LIN {X 0,Y 312.808,Z 286.335,A -85,B 0,C 180,E1 -15472.26,E2 -15472.26} C_VEL
LIN {X 0,Y 312.679,Z 286.347,A -85,B 0,C 180,E1 -15474.849,E2 -15474.849} C_VEL
LIN {X 0,Y 312.966,Z 286.313,A -85,B 0,C 180,E1 -15478.72,E2 -15478.72} C_VEL
LIN {X 0,Y 312.908,Z 286.323,A -85,B 0,C 180,E1 -15482.581,E2 -15482.581} C_VEL
LIN {X 0,Y 312.829,Z 286.33,A -85,B 0,C 180,E1 -15486.456,E2 -15486.456} C_VEL
LIN {X 0,Y 312.739,Z 286.341,A -85,B 0,C 180,E1 -15489.057,E2 -15489.057} C_VEL
LIN {X 0,Y 312.615,Z 286.358,A -85,B 0,C 180,E1 -15492.998,E2 -15492.998} C_VEL
LIN {X 0,Y 312.562,Z 286.36,A -85,B 0,C 180,E1 -15495.659,E2 -15495.659} C_VEL
LIN {X 0,Y 312.528,Z 286.365,A -85,B 0,C 180,E1 -15499.719,E2 -15499.719} C_VEL
LIN {X 0,Y 312.509,Z 286.369,A -85,B 0,C 180,E1 -15502.781,E2 -15502.781} C_VEL
LIN {X 0,Y 312.484,Z 286.371,A -85,B 0,C 180,E1 -15506.737,E2 -15506.737} C_VEL
LIN {X 0,Y 312.494,Z 286.371,A -85,B 0,C 180,E1 -15509.661,E2 -15509.661} C_VEL
LIN {X 0,Y 312.52,Z 286.369,A -85,B 0,C 180,E1 -15513.694,E2 -15513.694} C_VEL
LIN {X 0,Y 312.51,Z 286.371,A -85,B 0,C 180,E1 -15517.393,E2 -15517.393} C_VEL
LIN {X 0,Y 312.442,Z 286.374,A -85,B 0,C 180,E1 -15520.722,E2 -15520.722} C_VEL
LIN {X 0,Y 312.452,Z 286.375,A -85,B 0,C 180,E1 -15524.215,E2 -15524.215} C_VEL
LIN {X 0,Y 312.458,Z 286.378,A -85,B 0,C 180,E1 -15527.93,E2 -15527.93} C_VEL
LIN {X 0,Y 312.482,Z 286.376,A -85,B 0,C 180,E1 -15531.929,E2 -15531.929} C_VEL
LIN {X 0,Y 312.536,Z 286.367,A -85,B 0,C 180,E1 -15534.224,E2 -15534.224} C_VEL
LIN {X 0,Y 312.508,Z 286.367,A -85,B 0,C 180,E1 -15537.337,E2 -15537.337} C_VEL
LIN {X 0,Y 312.491,Z 286.369,A -85,B 0,C 180,E1 -15541.304,E2 -15541.304} C_VEL
LIN {X 0,Y 312.68,Z 286.545,A -85,B 0,C 180,E1 -15543.7,E2 -15543.7} C_VEL
LIN {X 0,Y 314.175,Z 295.332,A -85,B 0,C 180,E1 -15546.522,E2 -15546.522} C_VEL
LIN {X 0,Y 313.298,Z 305.478,A -85,B 0,C 180,E1 -15549.656,E2 -15549.656} C_VEL
LIN {X 0,Y 312.436,Z 315.736,A -85,B 0,C 180,E1 -15552.789,E2 -15552.789} C_VEL
LIN {X 0,Y 313.543,Z 332.693,A -85,B 0,C 180,E1 -15553.393,E2 -15553.393} C_VEL
LIN {X 0,Y 314.974,Z 349.181,A -85,B 0,C 180,E1 -15553.982,E2 -15553.982} C_VEL
LIN {X 0,Y 313.99,Z 394.354,A -85,B 0,C 180,E1 -15555.542,E2 -15555.542} C_VEL
LIN {X 0,Y 313.569,Z 406.833,A -85,B 0,C 180,E1 -15556.226,E2 -15556.226} C_VEL
LIN {X 0,Y 313.016,Z 417.039,A -85,B 0,C 180,E1 -15557.027,E2 -15557.027} C_VEL
LIN {X 0,Y 312.578,Z 425.178,A -85,B 0,C 180,E1 -15557.834,E2 -15557.834} C_VEL
LIN {X 0,Y 312.139,Z 433.195,A -85,B 0,C 180,E1 -15558.805,E2 -15558.805} C_VEL
LIN {X 0,Y 311.741,Z 441.983,A -85,B 0,C 180,E1 -15560.104,E2 -15560.104} C_VEL
LIN {X 0,Y 311.412,Z 449.886,A -85,B 0,C 180,E1 -15561.567,E2 -15561.567} C_VEL
LIN {X 0,Y 311.172,Z 456.813,A -85,B 0,C 180,E1 -15563.192,E2 -15563.192} C_VEL
LIN {X 0,Y 311.051,Z 460.872,A -85,B 0,C 180,E1 -15564.339,E2 -15564.339} C_VEL
LIN {X 0,Y 310.982,Z 464.265,A -85,B 0,C 180,E1 -15565.466,E2 -15565.466} C_VEL
LIN {X 0,Y 310.82,Z 468.668,A -85,B 0,C 180,E1 -15567.41,E2 -15567.41} C_VEL
LIN {X 0,Y 310.924,Z 470.88,A -85,B 0,C 180,E1 -15568.707,E2 -15568.707} C_VEL
LIN {X 0,Y 311.031,Z 472.489,A -85,B 0,C 180,E1 -15570.002,E2 -15570.002} C_VEL
LIN {X 0,Y 310.703,Z 473.409,A -85,B 0,C 180,E1 -15571.298,E2 -15571.298} C_VEL
LIN {X 0,Y 310.703,Z 473.802,A -85,B 0,C 180,E1 -15572.595,E2 -15572.595} C_VEL
LIN {X 0,Y 310.758,Z 473.691,A -85,B 0,C 180,E1 -15573.892,E2 -15573.892} C_VEL
LIN {X 0,Y 310.897,Z 472.45,A -85,B 0,C 180,E1 -15575.902,E2 -15575.902} C_VEL
LIN {X 0,Y 311.304,Z 470.124,A -85,B 0,C 180,E1 -15577.787,E2 -15577.787} C_VEL
LIN {X 0,Y 312.084,Z 466.493,A -85,B 0,C 180,E1 -15579.726,E2 -15579.726} C_VEL
LIN {X 0,Y 313.249,Z 461.354,A -85,B 0,C 180,E1 -15581.651,E2 -15581.651} C_VEL
LIN {X 0,Y 314.485,Z 455.869,A -85,B 0,C 180,E1 -15583.244,E2 -15583.244} C_VEL
LIN {X 0,Y 315.901,Z 449.073,A -85,B 0,C 180,E1 -15584.826,E2 -15584.826} C_VEL
LIN {X 0,Y 317.87,Z 439.738,A -85,B 0,C 180,E1 -15586.541,E2 -15586.541} C_VEL
LIN {X 0,Y 319.594,Z 431.167,A -85,B 0,C 180,E1 -15587.767,E2 -15587.767} C_VEL
LIN {X 0,Y 321.226,Z 422.026,A -85,B 0,C 180,E1 -15588.829,E2 -15588.829} C_VEL
LIN {X 0,Y 323.179,Z 410.428,A -85,B 0,C 180,E1 -15589.866,E2 -15589.866} C_VEL
LIN {X 0,Y 324.712,Z 399.087,A -85,B 0,C 180,E1 -15590.594,E2 -15590.594} C_VEL
LIN {X 0,Y 325.906,Z 386.794,A -85,B 0,C 180,E1 -15591.176,E2 -15591.176} C_VEL
LIN {X 0,Y 328.411,Z 352.215,A -85,B 0,C 180,E1 -15592.473,E2 -15592.473} C_VEL
LIN {X 0,Y 326.923,Z 339.744,A -85,B 0,C 180,E1 -15593.305,E2 -15593.305} C_VEL
LIN {X 0,Y 324.202,Z 325.651,A -85,B 0,C 180,E1 -15594.496,E2 -15594.496} C_VEL
LIN {X 0,Y 321.224,Z 313.546,A -85,B 0,C 180,E1 -15595.703,E2 -15595.703} C_VEL
LIN {X 0,Y 319.041,Z 308.853,A -85,B 0,C 180,E1 -15596.4,E2 -15596.4} C_VEL
LIN {X 0,Y 317.388,Z 301.3,A -85,B 0,C 180,E1 -15599.155,E2 -15599.155} C_VEL
LIN {X 0,Y 315.056,Z 293.728,A -85,B 0,C 180,E1 -15602.371,E2 -15602.371} C_VEL
LIN {X 0,Y 312.535,Z 286.365,A -85,B 0,C 180,E1 -15606.212,E2 -15606.212} C_VEL
LIN {X 0,Y 312.457,Z 286.373,A -85,B 0,C 180,E1 -15610.109,E2 -15610.109} C_VEL
LIN {X 0,Y 312.457,Z 286.374,A -85,B 0,C 180,E1 -15614.211,E2 -15614.211} C_VEL
LIN {X 0,Y 312.446,Z 286.373,A -85,B 0,C 180,E1 -15617.929,E2 -15617.929} C_VEL
LIN {X 0,Y 312.495,Z 286.365,A -85,B 0,C 180,E1 -15621.922,E2 -15621.922} C_VEL
LIN {X 0,Y 312.549,Z 286.361,A -85,B 0,C 180,E1 -15624.217,E2 -15624.217} C_VEL
LIN {X 0,Y 312.521,Z 286.366,A -85,B 0,C 180,E1 -15627.33,E2 -15627.33} C_VEL
LIN {X 0,Y 312.542,Z 286.523,A -85,B 0,C 180,E1 -15629.038,E2 -15629.038} C_VEL
LIN {X 0,Y 314.433,Z 291.517,A -85,B 0,C 180,E1 -15631.525,E2 -15631.525} C_VEL
LIN {X 0,Y 315.715,Z 294.654,A -85,B 0,C 180,E1 -15632.848,E2 -15632.848} C_VEL
LIN {X 0,Y 320.679,Z 302.089,A -85,B 0,C 180,E1 -15634.363,E2 -15634.363} C_VEL
LIN {X 0,Y 325.742,Z 310.91,A -85,B 0,C 180,E1 -15635.813,E2 -15635.813} C_VEL
LIN {X 0,Y 330.204,Z 320.269,A -85,B 0,C 180,E1 -15637.053,E2 -15637.053} C_VEL
LIN {X 0,Y 330.37,Z 321.468,A -85,B 0,C 180,E1 -15637.137,E2 -15637.137} C_VEL
LIN {X 0,Y 326.132,Z 374.77,A -85,B 0,C 180,E1 -15639.166,E2 -15639.166} C_VEL
LIN {X 0,Y 324.812,Z 387.33,A -85,B 0,C 180,E1 -15639.905,E2 -15639.905} C_VEL
LIN {X 0,Y 323.647,Z 396.64,A -85,B 0,C 180,E1 -15640.656,E2 -15640.656} C_VEL
LIN {X 0,Y 322.303,Z 405.621,A -85,B 0,C 180,E1 -15641.562,E2 -15641.562} C_VEL
LIN {X 0,Y 320.632,Z 415.281,A -85,B 0,C 180,E1 -15642.782,E2 -15642.782} C_VEL
LIN {X 0,Y 319.098,Z 422.949,A -85,B 0,C 180,E1 -15644.014,E2 -15644.014} C_VEL
LIN {X 0,Y 317.777,Z 429.28,A -85,B 0,C 180,E1 -15645.26,E2 -15645.26} C_VEL
LIN {X 0,Y 316.19,Z 435.818,A -85,B 0,C 180,E1 -15646.825,E2 -15646.825} C_VEL
LIN {X 0,Y 314.829,Z 441.072,A -85,B 0,C 180,E1 -15648.404,E2 -15648.404} C_VEL
LIN {X 0,Y 313.901,Z 444.428,A -85,B 0,C 180,E1 -15649.676,E2 -15649.676} C_VEL
LIN {X 0,Y 313.26,Z 447.125,A -85,B 0,C 180,E1 -15650.959,E2 -15650.959} C_VEL
LIN {X 0,Y 312.448,Z 449.278,A -85,B 0,C 180,E1 -15652.238,E2 -15652.238} C_VEL
LIN {X 0,Y 311.829,Z 450.845,A -85,B 0,C 180,E1 -15653.523,E2 -15653.523} C_VEL
LIN {X 0,Y 311.53,Z 451.786,A -85,B 0,C 180,E1 -15654.816,E2 -15654.816} C_VEL
LIN {X 0,Y 311.246,Z 452.205,A -85,B 0,C 180,E1 -15656.109,E2 -15656.109} C_VEL
LIN {X 0,Y 310.975,Z 452.125,A -85,B 0,C 180,E1 -15657.403,E2 -15657.403} C_VEL
LIN {X 0,Y 310.798,Z 451.534,A -85,B 0,C 180,E1 -15658.698,E2 -15658.698} C_VEL
LIN {X 0,Y 310.737,Z 450.385,A -85,B 0,C 180,E1 -15659.993,E2 -15659.993} C_VEL
LIN {X 0,Y 310.733,Z 447.533,A -85,B 0,C 180,E1 -15661.938,E2 -15661.938} C_VEL
LIN {X 0,Y 310.866,Z 444.951,A -85,B 0,C 180,E1 -15663.233,E2 -15663.233} C_VEL
LIN {X 0,Y 310.987,Z 441.657,A -85,B 0,C 180,E1 -15664.53,E2 -15664.53} C_VEL
LIN {X 0,Y 311.148,Z 435.238,A -85,B 0,C 180,E1 -15666.478,E2 -15666.478} C_VEL
LIN {X 0,Y 311.464,Z 429.92,A -85,B 0,C 180,E1 -15667.774,E2 -15667.774} C_VEL
LIN {X 0,Y 311.765,Z 423.504,A -85,B 0,C 180,E1 -15669.072,E2 -15669.072} C_VEL
LIN {X 0,Y 312.089,Z 415.727,A -85,B 0,C 180,E1 -15670.372,E2 -15670.372} C_VEL
LIN {X 0,Y 312.707,Z 406.255,A -85,B 0,C 180,E1 -15671.663,E2 -15671.663} C_VEL
LIN {X 0,Y 313.162,Z 395.383,A -85,B 0,C 180,E1 -15672.797,E2 -15672.797} C_VEL
LIN {X 0,Y 313.618,Z 385.414,A -85,B 0,C 180,E1 -15673.602,E2 -15673.602} C_VEL
LIN {X 0,Y 313.997,Z 373.275,A -85,B 0,C 180,E1 -15674.328,E2 -15674.328} C_VEL
LIN {X 0,Y 314.475,Z 353.255,A -85,B 0,C 180,E1 -15675.051,E2 -15675.051} C_VEL
LIN {X 0,Y 315.258,Z 313.185,A -85,B 0,C 180,E1 -15676.405,E2 -15676.405} C_VEL
LIN {X 0,Y 312.719,Z 292.458,A -85,B 0,C 180,E1 -15677.169,E2 -15677.169} C_VEL
LIN {X 0,Y 312.756,Z 286.337,A -85,B 0,C 180,E1 -15679.323,E2 -15679.323} C_VEL
LIN {X 0,Y 312.478,Z 286.373,A -85,B 0,C 180,E1 -15683.873,E2 -15683.873} C_VEL
LIN {X 0,Y 312.468,Z 286.373,A -85,B 0,C 180,E1 -15686.724,E2 -15686.724} C_VEL
LIN {X 0,Y 312.451,Z 286.374,A -85,B 0,C 180,E1 -15689.65,E2 -15689.65} C_VEL
LIN {X 0,Y 312.501,Z 286.368,A -85,B 0,C 180,E1 -15693.681,E2 -15693.681} C_VEL
LIN {X 0,Y 312.491,Z 286.369,A -85,B 0,C 180,E1 -15697.379,E2 -15697.379} C_VEL
LIN {X 0,Y 312.415,Z 286.383,A -85,B 0,C 180,E1 -15700.71,E2 -15700.71} C_VEL
LIN {X 0,Y 312.423,Z 286.379,A -85,B 0,C 180,E1 -15704.203,E2 -15704.203} C_VEL
LIN {X 0,Y 312.437,Z 286.375,A -85,B 0,C 180,E1 -15707.915,E2 -15707.915} C_VEL
LIN {X 0,Y 312.464,Z 286.378,A -85,B 0,C 180,E1 -15710.964,E2 -15710.964} C_VEL
LIN {X 0,Y 312.495,Z 286.368,A -85,B 0,C 180,E1 -15714.213,E2 -15714.213} C_VEL
LIN {X 0,Y 312.463,Z 286.375,A -85,B 0,C 180,E1 -15717.327,E2 -15717.327} C_VEL
LIN {X 0,Y 312.526,Z 286.365,A -85,B 0,C 180,E1 -15721.818,E2 -15721.818} C_VEL
LIN {X 0,Y 312.541,Z 286.363,A -85,B 0,C 180,E1 -15724.705,E2 -15724.705} C_VEL
LIN {X 0,Y 312.522,Z 286.369,A -85,B 0,C 180,E1 -15727.522,E2 -15727.522} C_VEL
LIN {X 0,Y 312.591,Z 286.361,A -85,B 0,C 180,E1 -15731.651,E2 -15731.651} C_VEL
LIN {X 0,Y 312.645,Z 286.354,A -85,B 0,C 180,E1 -15735.682,E2 -15735.682} C_VEL
LIN {X 0,Y 312.652,Z 286.354,A -85,B 0,C 180,E1 -15739.638,E2 -15739.638} C_VEL
LIN {X 0,Y 312.81,Z 286.331,A -85,B 0,C 180,E1 -15742.251,E2 -15742.251} C_VEL
LIN {X 0,Y 312.67,Z 286.346,A -85,B 0,C 180,E1 -15744.839,E2 -15744.839} C_VEL
LIN {X 0,Y 312.908,Z 286.318,A -85,B 0,C 180,E1 -15747.423,E2 -15747.423} C_VEL
LIN {X 0,Y 313.067,Z 286.303,A -85,B 0,C 180,E1 -15749.998,E2 -15749.998} C_VEL
LIN {X 0,Y 312.906,Z 286.318,A -85,B 0,C 180,E1 -15752.572,E2 -15752.572} C_VEL
LIN {X 0,Y 312.849,Z 286.327,A -85,B 0,C 180,E1 -15756.447,E2 -15756.447} C_VEL
LIN {X 0,Y 312.732,Z 286.339,A -85,B 0,C 180,E1 -15759.048,E2 -15759.048} C_VEL
LIN {X 0,Y 312.581,Z 286.358,A -85,B 0,C 180,E1 -15762.991,E2 -15762.991} C_VEL
LIN {X 0,Y 312.575,Z 286.358,A -85,B 0,C 180,E1 -15765.65,E2 -15765.65} C_VEL
LIN {X 0,Y 312.554,Z 286.361,A -85,B 0,C 180,E1 -15769.225,E2 -15769.225} C_VEL
LIN {X 0,Y 312.475,Z 286.375,A -85,B 0,C 180,E1 -15772.782,E2 -15772.782} C_VEL
LIN {X 0,Y 312.544,Z 286.362,A -85,B 0,C 180,E1 -15775.935,E2 -15775.935} C_VEL
LIN {X 0,Y 312.493,Z 286.368,A -85,B 0,C 180,E1 -15779.652,E2 -15779.652} C_VEL
LIN {X 0,Y 312.469,Z 286.372,A -85,B 0,C 180,E1 -15783.692,E2 -15783.692} C_VEL
LIN {X 0,Y 312.492,Z 286.371,A -85,B 0,C 180,E1 -15787.386,E2 -15787.386} C_VEL
LIN {X 0,Y 312.481,Z 286.372,A -85,B 0,C 180,E1 -15790.707,E2 -15790.707} C_VEL
LIN {X 0,Y 312.549,Z 286.361,A -85,B 0,C 180,E1 -15794.188,E2 -15794.188} C_VEL
LIN {X 0,Y 312.513,Z 286.367,A -85,B 0,C 180,E1 -15797.909,E2 -15797.909} C_VEL
LIN {X 0,Y 312.502,Z 286.369,A -85,B 0,C 180,E1 -15801.914,E2 -15801.914} C_VEL
LIN {X 0,Y 312.467,Z 286.375,A -85,B 0,C 180,E1 -15805.795,E2 -15805.795} C_VEL
LIN {X 0,Y 312.483,Z 286.37,A -85,B 0,C 180,E1 -15808.859,E2 -15808.859} C_VEL
LIN {X 0,Y 312.535,Z 286.368,A -85,B 0,C 180,E1 -15811.83,E2 -15811.83} C_VEL
LIN {X 0,Y 312.551,Z 286.361,A -85,B 0,C 180,E1 -15814.717,E2 -15814.717} C_VEL
LIN {X 0,Y 312.499,Z 286.367,A -85,B 0,C 180,E1 -15818.015,E2 -15818.015} C_VEL
LIN {X 0,Y 312.538,Z 286.366,A -85,B 0,C 180,E1 -15821.658,E2 -15821.658} C_VEL
LIN {X 0,Y 312.553,Z 286.36,A -85,B 0,C 180,E1 -15823.623,E2 -15823.623} C_VEL
LIN {X 0,Y 311.906,Z 286.444,A -85,B 0,C 180,E1 -15824.699,E2 -15824.699} C_VEL
LIN {X 0,Y 309.047,Z 286.8,A -85,B 0,C 180,E1 -15826.449,E2 -15826.449} C_VEL
LIN {X 0,Y 306.64,Z 287.1,A -85,B 0,C 180,E1 -15827.869,E2 -15827.869} C_VEL
LIN {X 0,Y 305.652,Z 287.221,A -85,B 0,C 180,E1 -15828.969,E2 -15828.969} C_VEL
LIN {X 0,Y 305.596,Z 287.228,A -85,B 0,C 180,E1 -15829.341,E2 -15829.341} C_VEL
LIN {X 0,Y 305.75,Z 287.212,A -85,B 0,C 180,E1 -15832.08,E2 -15832.08} C_VEL
LIN {X 0,Y 305.649,Z 287.223,A -85,B 0,C 180,E1 -15834.73,E2 -15834.73} C_VEL
LIN {X 0,Y 305.933,Z 287.189,A -85,B 0,C 180,E1 -15838.69,E2 -15838.69} C_VEL
LIN {X 0,Y 305.923,Z 287.187,A -85,B 0,C 180,E1 -15841.323,E2 -15841.323} C_VEL
LIN {X 0,Y 305.652,Z 287.221,A -85,B 0,C 180,E1 -15845.284,E2 -15845.284} C_VEL
LIN {X 0,Y 305.734,Z 287.211,A -85,B 0,C 180,E1 -15847.934,E2 -15847.934} C_VEL
LIN {X 0,Y 305.585,Z 287.229,A -85,B 0,C 180,E1 -15851.952,E2 -15851.952} C_VEL
LIN {X 0,Y 305.551,Z 287.238,A -85,B 0,C 180,E1 -15854.985,E2 -15854.985} C_VEL
LIN {X 0,Y 305.502,Z 287.243,A -85,B 0,C 180,E1 -15858.794,E2 -15858.794} C_VEL
LIN {X 0,Y 305.452,Z 287.25,A -85,B 0,C 180,E1 -15863.032,E2 -15863.032} C_VEL
LIN {X 0,Y 305.45,Z 287.246,A -85,B 0,C 180,E1 -15866.197,E2 -15866.197} C_VEL
LIN {X 0,Y 305.447,Z 287.25,A -85,B 0,C 180,E1 -15869.039,E2 -15869.039} C_VEL
LIN {X 0,Y 305.436,Z 287.248,A -85,B 0,C 180,E1 -15871.959,E2 -15871.959} C_VEL
LIN {X 0,Y 305.461,Z 287.247,A -85,B 0,C 180,E1 -15875.119,E2 -15875.119} C_VEL
LIN {X 0,Y 305.436,Z 287.247,A -85,B 0,C 180,E1 -15878.53,E2 -15878.53} C_VEL
LIN {X 0,Y 305.436,Z 287.247,A -85,B 0,C 180,E1 -15882.586,E2 -15882.586} C_VEL
LIN {X 0,Y 305.424,Z 287.25,A -85,B 0,C 180,E1 -15886.349,E2 -15886.349} C_VEL
LIN {X 0,Y 305.415,Z 287.255,A -85,B 0,C 180,E1 -15889.889,E2 -15889.889} C_VEL
LIN {X 0,Y 305.467,Z 287.246,A -85,B 0,C 180,E1 -15893.642,E2 -15893.642} C_VEL
LIN {X 0,Y 305.472,Z 287.245,A -85,B 0,C 180,E1 -15896.487,E2 -15896.487} C_VEL
LIN {X 0,Y 305.424,Z 287.25,A -85,B 0,C 180,E1 -15899.59,E2 -15899.59} C_VEL
LIN {X 0,Y 305.616,Z 287.307,A -85,B 0,C 180,E1 -15903.638,E2 -15903.638} C_VEL
LIN {X 0,Y 307.022,Z 295.41,A -85,B 0,C 180,E1 -15906.305,E2 -15906.305} C_VEL
LIN {X 0,Y 306.69,Z 301.192,A -85,B 0,C 180,E1 -15908.14,E2 -15908.14} C_VEL
LIN {X 0,Y 305.38,Z 315.452,A -85,B 0,C 180,E1 -15912.636,E2 -15912.636} C_VEL
LIN {X 0,Y 306.378,Z 331.761,A -85,B 0,C 180,E1 -15913.238,E2 -15913.238} C_VEL
LIN {X 0,Y 307.903,Z 349.63,A -85,B 0,C 180,E1 -15913.902,E2 -15913.902} C_VEL
LIN {X 0,Y 306.913,Z 394.247,A -85,B 0,C 180,E1 -15915.498,E2 -15915.498} C_VEL
LIN {X 0,Y 306.468,Z 407.18,A -85,B 0,C 180,E1 -15916.239,E2 -15916.239} C_VEL
LIN {X 0,Y 305.919,Z 417.254,A -85,B 0,C 180,E1 -15917.059,E2 -15917.059} C_VEL
LIN {X 0,Y 305.357,Z 426.75,A -85,B 0,C 180,E1 -15918.048,E2 -15918.048} C_VEL
LIN {X 0,Y 304.903,Z 436.813,A -85,B 0,C 180,E1 -15919.376,E2 -15919.376} C_VEL
LIN {X 0,Y 304.526,Z 444.734,A -85,B 0,C 180,E1 -15920.706,E2 -15920.706} C_VEL
LIN {X 0,Y 304.281,Z 451.287,A -85,B 0,C 180,E1 -15922.037,E2 -15922.037} C_VEL
LIN {X 0,Y 304.097,Z 456.716,A -85,B 0,C 180,E1 -15923.367,E2 -15923.367} C_VEL
LIN {X 0,Y 303.996,Z 461.21,A -85,B 0,C 180,E1 -15924.696,E2 -15924.696} C_VEL
LIN {X 0,Y 303.844,Z 464.871,A -85,B 0,C 180,E1 -15926.023,E2 -15926.023} C_VEL
LIN {X 0,Y 303.808,Z 469.028,A -85,B 0,C 180,E1 -15928.014,E2 -15928.014} C_VEL
LIN {X 0,Y 303.842,Z 470.176,A -85,B 0,C 180,E1 -15928.677,E2 -15928.677} C_VEL
LIN {X 0,Y 303.97,Z 471.84,A -85,B 0,C 180,E1 -15930.002,E2 -15930.002} C_VEL
LIN {X 0,Y 303.622,Z 472.879,A -85,B 0,C 180,E1 -15931.329,E2 -15931.329} C_VEL
LIN {X 0,Y 303.628,Z 473.429,A -85,B 0,C 180,E1 -15932.656,E2 -15932.656} C_VEL
LIN {X 0,Y 303.675,Z 473.472,A -85,B 0,C 180,E1 -15933.983,E2 -15933.983} C_VEL
LIN {X 0,Y 303.792,Z 472.565,A -85,B 0,C 180,E1 -15935.827,E2 -15935.827} C_VEL
LIN {X 0,Y 304.276,Z 470.237,A -85,B 0,C 180,E1 -15937.968,E2 -15937.968} C_VEL
LIN {X 0,Y 305.086,Z 466.811,A -85,B 0,C 180,E1 -15939.951,E2 -15939.951} C_VEL
LIN {X 0,Y 306.341,Z 461.995,A -85,B 0,C 180,E1 -15941.918,E2 -15941.918} C_VEL
LIN {X 0,Y 307.933,Z 455.501,A -85,B 0,C 180,E1 -15943.868,E2 -15943.868} C_VEL
LIN {X 0,Y 309.143,Z 450.242,A -85,B 0,C 180,E1 -15945.158,E2 -15945.158} C_VEL
LIN {X 0,Y 310.569,Z 443.978,A -85,B 0,C 180,E1 -15946.433,E2 -15946.433} C_VEL
LIN {X 0,Y 312.312,Z 436.428,A -85,B 0,C 180,E1 -15947.688,E2 -15947.688} C_VEL
LIN {X 0,Y 314.229,Z 427.283,A -85,B 0,C 180,E1 -15948.925,E2 -15948.925} C_VEL
LIN {X 0,Y 316.098,Z 417.336,A -85,B 0,C 180,E1 -15949.991,E2 -15949.991} C_VEL
LIN {X 0,Y 317.921,Z 406.353,A -85,B 0,C 180,E1 -15950.885,E2 -15950.885} C_VEL
LIN {X 0,Y 319.594,Z 394.24,A -85,B 0,C 180,E1 -15951.615,E2 -15951.615} C_VEL
LIN {X 0,Y 321.622,Z 369.527,A -85,B 0,C 180,E1 -15952.6,E2 -15952.6} C_VEL
LIN {X 0,Y 322.874,Z 353.385,A -85,B 0,C 180,E1 -15953.232,E2 -15953.232} C_VEL
LIN {X 0,Y 321.463,Z 340.839,A -85,B 0,C 180,E1 -15954.132,E2 -15954.132} C_VEL
LIN {X 0,Y 318.87,Z 327.161,A -85,B 0,C 180,E1 -15955.35,E2 -15955.35} C_VEL
LIN {X 0,Y 316.464,Z 317.354,A -85,B 0,C 180,E1 -15956.404,E2 -15956.404} C_VEL
LIN {X 0,Y 314.296,Z 312.894,A -85,B 0,C 180,E1 -15957.128,E2 -15957.128} C_VEL
LIN {X 0,Y 311.945,Z 308.011,A -85,B 0,C 180,E1 -15958.032,E2 -15958.032} C_VEL
LIN {X 0,Y 310.884,Z 303.44,A -85,B 0,C 180,E1 -15959.826,E2 -15959.826} C_VEL
LIN {X 0,Y 308.965,Z 297.154,A -85,B 0,C 180,E1 -15962.68,E2 -15962.68} C_VEL
LIN {X 0,Y 307.021,Z 291.567,A -85,B 0,C 180,E1 -15965.715,E2 -15965.715} C_VEL
LIN {X 0,Y 305.449,Z 287.248,A -85,B 0,C 180,E1 -15968.677,E2 -15968.677} C_VEL
LIN {X 0,Y 305.419,Z 287.253,A -85,B 0,C 180,E1 -15972.572,E2 -15972.572} C_VEL
LIN {X 0,Y 305.421,Z 287.25,A -85,B 0,C 180,E1 -15976.338,E2 -15976.338} C_VEL
LIN {X 0,Y 305.428,Z 287.246,A -85,B 0,C 180,E1 -15979.882,E2 -15979.882} C_VEL
LIN {X 0,Y 305.481,Z 287.24,A -85,B 0,C 180,E1 -15983.634,E2 -15983.634} C_VEL
LIN {X 0,Y 305.486,Z 287.248,A -85,B 0,C 180,E1 -15986.48,E2 -15986.48} C_VEL
LIN {X 0,Y 307.066,Z 291.123,A -85,B 0,C 180,E1 -15988.999,E2 -15988.999} C_VEL
LIN {X 0,Y 308.688,Z 295.341,A -85,B 0,C 180,E1 -15991.171,E2 -15991.171} C_VEL
LIN {X 0,Y 315.081,Z 304.674,A -85,B 0,C 180,E1 -15993.37,E2 -15993.37} C_VEL
LIN {X 0,Y 319.786,Z 312.784,A -85,B 0,C 180,E1 -15994.832,E2 -15994.832} C_VEL
LIN {X 0,Y 324.2,Z 321.551,A -85,B 0,C 180,E1 -15996.13,E2 -15996.13} C_VEL
LIN {X 0,Y 325.013,Z 323.476,A -85,B 0,C 180,E1 -15996.372,E2 -15996.372} C_VEL
LIN {X 0,Y 320.464,Z 375.997,A -85,B 0,C 180,E1 -15998.443,E2 -15998.443} C_VEL
LIN {X 0,Y 319.046,Z 388.238,A -85,B 0,C 180,E1 -15999.188,E2 -15999.188} C_VEL
LIN {X 0,Y 317.797,Z 397.34,A -85,B 0,C 180,E1 -15999.948,E2 -15999.948} C_VEL
LIN {X 0,Y 316.137,Z 407.489,A -85,B 0,C 180,E1 -16001.021,E2 -16001.021} C_VEL
LIN {X 0,Y 314.085,Z 417.682,A -85,B 0,C 180,E1 -16002.412,E2 -16002.412} C_VEL
LIN {X 0,Y 312.509,Z 425.008,A -85,B 0,C 180,E1 -16003.668,E2 -16003.668} C_VEL
LIN {X 0,Y 311.114,Z 431.083,A -85,B 0,C 180,E1 -16004.937,E2 -16004.937} C_VEL
LIN {X 0,Y 309.755,Z 436.186,A -85,B 0,C 180,E1 -16006.212,E2 -16006.212} C_VEL
LIN {X 0,Y 308.565,Z 440.441,A -85,B 0,C 180,E1 -16007.498,E2 -16007.498} C_VEL
LIN {X 0,Y 307,Z 445.503,A -85,B 0,C 180,E1 -16009.441,E2 -16009.441} C_VEL
LIN {X 0,Y 306.322,Z 448.021,A -85,B 0,C 180,E1 -16010.752,E2 -16010.752} C_VEL
LIN {X 0,Y 305.468,Z 450.005,A -85,B 0,C 180,E1 -16012.059,E2 -16012.059} C_VEL
LIN {X 0,Y 304.819,Z 451.444,A -85,B 0,C 180,E1 -16013.374,E2 -16013.374} C_VEL
LIN {X 0,Y 304.479,Z 452.315,A -85,B 0,C 180,E1 -16014.696,E2 -16014.696} C_VEL
LIN {X 0,Y 304.178,Z 452.582,A -85,B 0,C 180,E1 -16016.019,E2 -16016.019} C_VEL
LIN {X 0,Y 303.897,Z 452.339,A -85,B 0,C 180,E1 -16017.342,E2 -16017.342} C_VEL
LIN {X 0,Y 303.712,Z 451.593,A -85,B 0,C 180,E1 -16018.667,E2 -16018.667} C_VEL
LIN {X 0,Y 303.649,Z 450.326,A -85,B 0,C 180,E1 -16019.993,E2 -16019.993} C_VEL
LIN {X 0,Y 303.653,Z 447.255,A -85,B 0,C 180,E1 -16021.983,E2 -16021.983} C_VEL
LIN {X 0,Y 303.898,Z 442.856,A -85,B 0,C 180,E1 -16023.971,E2 -16023.971} C_VEL
LIN {X 0,Y 303.965,Z 436.98,A -85,B 0,C 180,E1 -16025.941,E2 -16025.941} C_VEL
LIN {X 0,Y 304.347,Z 430.388,A -85,B 0,C 180,E1 -16027.623,E2 -16027.623} C_VEL
LIN {X 0,Y 304.632,Z 424.032,A -85,B 0,C 180,E1 -16028.952,E2 -16028.952} C_VEL
LIN {X 0,Y 305.026,Z 416.328,A -85,B 0,C 180,E1 -16030.279,E2 -16030.279} C_VEL
LIN {X 0,Y 305.564,Z 406.898,A -85,B 0,C 180,E1 -16031.603,E2 -16031.603} C_VEL
LIN {X 0,Y 306.042,Z 396.182,A -85,B 0,C 180,E1 -16032.762,E2 -16032.762} C_VEL
LIN {X 0,Y 306.503,Z 386.353,A -85,B 0,C 180,E1 -16033.586,E2 -16033.586} C_VEL
LIN {X 0,Y 306.882,Z 375.278,A -85,B 0,C 180,E1 -16034.287,E2 -16034.287} C_VEL
LIN {X 0,Y 307.226,Z 359.888,A -85,B 0,C 180,E1 -16034.905,E2 -16034.905} C_VEL
LIN {X 0,Y 308.152,Z 313.414,A -85,B 0,C 180,E1 -16036.525,E2 -16036.525} C_VEL
LIN {X 0,Y 305.682,Z 292.925,A -85,B 0,C 180,E1 -16037.304,E2 -16037.304} C_VEL
LIN {X 0,Y 305.714,Z 287.215,A -85,B 0,C 180,E1 -16039.284,E2 -16039.284} C_VEL
LIN {X 0,Y 305.443,Z 287.25,A -85,B 0,C 180,E1 -16044.458,E2 -16044.458} C_VEL
LIN {X 0,Y 305.426,Z 287.249,A -85,B 0,C 180,E1 -16047.391,E2 -16047.391} C_VEL
LIN {X 0,Y 305.4,Z 287.257,A -85,B 0,C 180,E1 -16050.406,E2 -16050.406} C_VEL
LIN {X 0,Y 305.445,Z 287.249,A -85,B 0,C 180,E1 -16054.07,E2 -16054.07} C_VEL
LIN {X 0,Y 305.431,Z 287.252,A -85,B 0,C 180,E1 -16056.735,E2 -16056.735} C_VEL
LIN {X 0,Y 305.384,Z 287.259,A -85,B 0,C 180,E1 -16060.582,E2 -16060.582} C_VEL
LIN {X 0,Y 305.394,Z 287.253,A -85,B 0,C 180,E1 -16063.649,E2 -16063.649} C_VEL
LIN {X 0,Y 305.411,Z 287.251,A -85,B 0,C 180,E1 -16067.41,E2 -16067.41} C_VEL
LIN {X 0,Y 305.426,Z 287.248,A -85,B 0,C 180,E1 -16069.885,E2 -16069.885} C_VEL
LIN {X 0,Y 305.444,Z 287.247,A -85,B 0,C 180,E1 -16073.625,E2 -16073.625} C_VEL
LIN {X 0,Y 305.427,Z 287.25,A -85,B 0,C 180,E1 -16076.476,E2 -16076.476} C_VEL
LIN {X 0,Y 305.439,Z 287.25,A -85,B 0,C 180,E1 -16080.95,E2 -16080.95} C_VEL
LIN {X 0,Y 305.521,Z 287.237,A -85,B 0,C 180,E1 -16084.081,E2 -16084.081} C_VEL
LIN {X 0,Y 305.436,Z 287.247,A -85,B 0,C 180,E1 -16088.396,E2 -16088.396} C_VEL
LIN {X 0,Y 305.533,Z 287.239,A -85,B 0,C 180,E1 -16091.212,E2 -16091.212} C_VEL
LIN {X 0,Y 305.59,Z 287.232,A -85,B 0,C 180,E1 -16095.344,E2 -16095.344} C_VEL
LIN {X 0,Y 305.589,Z 287.231,A -85,B 0,C 180,E1 -16099.396,E2 -16099.396} C_VEL
LIN {X 0,Y 305.753,Z 287.211,A -85,B 0,C 180,E1 -16102.071,E2 -16102.071} C_VEL
LIN {X 0,Y 305.64,Z 287.222,A -85,B 0,C 180,E1 -16104.72,E2 -16104.72} C_VEL
LIN {X 0,Y 305.91,Z 287.189,A -85,B 0,C 180,E1 -16108.681,E2 -16108.681} C_VEL
LIN {X 0,Y 305.91,Z 287.189,A -85,B 0,C 180,E1 -16111.314,E2 -16111.314} C_VEL
LIN {X 0,Y 305.637,Z 287.222,A -85,B 0,C 180,E1 -16115.275,E2 -16115.275} C_VEL
LIN {X 0,Y 305.749,Z 287.212,A -85,B 0,C 180,E1 -16117.925,E2 -16117.925} C_VEL
LIN {X 0,Y 305.551,Z 287.235,A -85,B 0,C 180,E1 -16121.945,E2 -16121.945} C_VEL
LIN {X 0,Y 305.567,Z 287.232,A -85,B 0,C 180,E1 -16125.023,E2 -16125.023} C_VEL
LIN {X 0,Y 305.525,Z 287.24,A -85,B 0,C 180,E1 -16128.784,E2 -16128.784} C_VEL
LIN {X 0,Y 305.434,Z 287.25,A -85,B 0,C 180,E1 -16133.041,E2 -16133.041} C_VEL
LIN {X 0,Y 305.474,Z 287.244,A -85,B 0,C 180,E1 -16136.22,E2 -16136.22} C_VEL
LIN {X 0,Y 305.444,Z 287.25,A -85,B 0,C 180,E1 -16139.052,E2 -16139.052} C_VEL
LIN {X 0,Y 305.415,Z 287.251,A -85,B 0,C 180,E1 -16143.52,E2 -16143.52} C_VEL
LIN {X 0,Y 305.448,Z 287.249,A -85,B 0,C 180,E1 -16146.74,E2 -16146.74} C_VEL
LIN {X 0,Y 305.44,Z 287.248,A -85,B 0,C 180,E1 -16150.61,E2 -16150.61} C_VEL
LIN {X 0,Y 305.499,Z 287.24,A -85,B 0,C 180,E1 -16154.521,E2 -16154.521} C_VEL
LIN {X 0,Y 305.457,Z 287.245,A -85,B 0,C 180,E1 -16158.158,E2 -16158.158} C_VEL
LIN {X 0,Y 305.468,Z 287.248,A -85,B 0,C 180,E1 -16161.607,E2 -16161.607} C_VEL
LIN {X 0,Y 305.423,Z 287.25,A -85,B 0,C 180,E1 -16164.892,E2 -16164.892} C_VEL
LIN {X 0,Y 305.412,Z 287.25,A -85,B 0,C 180,E1 -16168.362,E2 -16168.362} C_VEL
LIN {X 0,Y 305.477,Z 287.243,A -85,B 0,C 180,E1 -16171.119,E2 -16171.119} C_VEL
LIN {X 0,Y 305.537,Z 287.238,A -85,B 0,C 180,E1 -16174.094,E2 -16174.094} C_VEL
LIN {X 0,Y 305.443,Z 287.248,A -85,B 0,C 180,E1 -16178.407,E2 -16178.407} C_VEL
LIN {X 0,Y 305.489,Z 287.241,A -85,B 0,C 180,E1 -16181.219,E2 -16181.219} C_VEL
LIN {X 0,Y 305.601,Z 287.227,A -85,B 0,C 180,E1 -16185.354,E2 -16185.354} C_VEL
LIN {X 0,Y 305.596,Z 287.228,A -85,B 0,C 180,E1 -16189.341,E2 -16189.341} C_VEL
LIN {X 0,Y 305.001,Z 287.306,A -85,B 0,C 180,E1 -16190.443,E2 -16190.443} C_VEL
LIN {X 0,Y 302.193,Z 287.657,A -85,B 0,C 180,E1 -16192.237,E2 -16192.237} C_VEL
LIN {X 0,Y 299.75,Z 287.959,A -85,B 0,C 180,E1 -16193.693,E2 -16193.693} C_VEL
LIN {X 0,Y 298.67,Z 288.092,A -85,B 0,C 180,E1 -16194.82,E2 -16194.82} C_VEL
LIN {X 0,Y 298.568,Z 288.102,A -85,B 0,C 180,E1 -16195.202,E2 -16195.202} C_VEL
LIN {X 0,Y 298.899,Z 288.066,A -85,B 0,C 180,E1 -16198.66,E2 -16198.66} C_VEL
LIN {X 0,Y 298.891,Z 288.063,A -85,B 0,C 180,E1 -16201.354,E2 -16201.354} C_VEL
LIN {X 0,Y 298.621,Z 288.096,A -85,B 0,C 180,E1 -16205.408,E2 -16205.408} C_VEL
LIN {X 0,Y 298.697,Z 288.092,A -85,B 0,C 180,E1 -16208.826,E2 -16208.826} C_VEL
LIN {X 0,Y 298.534,Z 288.108,A -85,B 0,C 180,E1 -16212.238,E2 -16212.238} C_VEL
LIN {X 0,Y 298.516,Z 288.113,A -85,B 0,C 180,E1 -16215.157,E2 -16215.157} C_VEL
LIN {X 0,Y 298.432,Z 288.121,A -85,B 0,C 180,E1 -16219.621,E2 -16219.621} C_VEL
LIN {X 0,Y 298.378,Z 288.128,A -85,B 0,C 180,E1 -16223.61,E2 -16223.61} C_VEL
LIN {X 0,Y 298.401,Z 288.125,A -85,B 0,C 180,E1 -16226.589,E2 -16226.589} C_VEL
LIN {X 0,Y 298.392,Z 288.127,A -85,B 0,C 180,E1 -16229.65,E2 -16229.65} C_VEL
LIN {X 0,Y 298.393,Z 288.125,A -85,B 0,C 180,E1 -16232.806,E2 -16232.806} C_VEL
LIN {X 0,Y 298.404,Z 288.125,A -85,B 0,C 180,E1 -16236.078,E2 -16236.078} C_VEL
LIN {X 0,Y 298.376,Z 288.132,A -85,B 0,C 180,E1 -16239.497,E2 -16239.497} C_VEL
LIN {X 0,Y 298.372,Z 288.128,A -85,B 0,C 180,E1 -16243.102,E2 -16243.102} C_VEL
LIN {X 0,Y 298.374,Z 288.127,A -85,B 0,C 180,E1 -16246.919,E2 -16246.919} C_VEL
LIN {X 0,Y 298.391,Z 288.125,A -85,B 0,C 180,E1 -16251.016,E2 -16251.016} C_VEL
LIN {X 0,Y 298.41,Z 288.128,A -85,B 0,C 180,E1 -16253.932,E2 -16253.932} C_VEL
LIN {X 0,Y 298.4,Z 288.124,A -85,B 0,C 180,E1 -16257.204,E2 -16257.204} C_VEL
LIN {X 0,Y 298.439,Z 288.122,A -85,B 0,C 180,E1 -16261.905,E2 -16261.905} C_VEL
LIN {X 0,Y 298.594,Z 288.276,A -85,B 0,C 180,E1 -16263.657,E2 -16263.657} C_VEL
LIN {X 0,Y 300.005,Z 296.834,A -85,B 0,C 180,E1 -16266.534,E2 -16266.534} C_VEL
LIN {X 0,Y 299.033,Z 307.031,A -85,B 0,C 180,E1 -16269.839,E2 -16269.839} C_VEL
LIN {X 0,Y 298.309,Z 315.184,A -85,B 0,C 180,E1 -16272.478,E2 -16272.478} C_VEL
LIN {X 0,Y 299.273,Z 331.823,A -85,B 0,C 180,E1 -16273.126,E2 -16273.126} C_VEL
LIN {X 0,Y 300.815,Z 349.751,A -85,B 0,C 180,E1 -16273.809,E2 -16273.809} C_VEL
LIN {X 0,Y 299.812,Z 394.099,A -85,B 0,C 180,E1 -16275.45,E2 -16275.45} C_VEL
LIN {X 0,Y 299.404,Z 406.413,A -85,B 0,C 180,E1 -16276.167,E2 -16276.167} C_VEL
LIN {X 0,Y 298.897,Z 415.678,A -85,B 0,C 180,E1 -16276.922,E2 -16276.922} C_VEL
LIN {X 0,Y 298.466,Z 423.95,A -85,B 0,C 180,E1 -16277.767,E2 -16277.767} C_VEL
LIN {X 0,Y 298.025,Z 432.038,A -85,B 0,C 180,E1 -16278.784,E2 -16278.784} C_VEL
LIN {X 0,Y 297.692,Z 439.858,A -85,B 0,C 180,E1 -16279.976,E2 -16279.976} C_VEL
LIN {X 0,Y 297.295,Z 448.087,A -85,B 0,C 180,E1 -16281.506,E2 -16281.506} C_VEL
LIN {X 0,Y 297.058,Z 455.277,A -85,B 0,C 180,E1 -16283.209,E2 -16283.209} C_VEL
LIN {X 0,Y 296.953,Z 459.964,A -85,B 0,C 180,E1 -16284.57,E2 -16284.57} C_VEL
LIN {X 0,Y 296.798,Z 463.821,A -85,B 0,C 180,E1 -16285.929,E2 -16285.929} C_VEL
LIN {X 0,Y 296.69,Z 466.932,A -85,B 0,C 180,E1 -16287.287,E2 -16287.287} C_VEL
LIN {X 0,Y 296.802,Z 469.354,A -85,B 0,C 180,E1 -16288.645,E2 -16288.645} C_VEL
LIN {X 0,Y 296.909,Z 471.149,A -85,B 0,C 180,E1 -16290.002,E2 -16290.002} C_VEL
LIN {X 0,Y 296.542,Z 472.348,A -85,B 0,C 180,E1 -16291.36,E2 -16291.36} C_VEL
LIN {X 0,Y 296.556,Z 473.054,A -85,B 0,C 180,E1 -16292.719,E2 -16292.719} C_VEL
LIN {X 0,Y 296.594,Z 473.23,A -85,B 0,C 180,E1 -16294.079,E2 -16294.079} C_VEL
LIN {X 0,Y 296.685,Z 472.66,A -85,B 0,C 180,E1 -16295.746,E2 -16295.746} C_VEL
LIN {X 0,Y 297.233,Z 470.364,A -85,B 0,C 180,E1 -16298.158,E2 -16298.158} C_VEL
LIN {X 0,Y 298.106,Z 467.102,A -85,B 0,C 180,E1 -16300.187,E2 -16300.187} C_VEL
LIN {X 0,Y 298.944,Z 464.22,A -85,B 0,C 180,E1 -16301.529,E2 -16301.529} C_VEL
LIN {X 0,Y 300.544,Z 458.677,A -85,B 0,C 180,E1 -16303.526,E2 -16303.526} C_VEL
LIN {X 0,Y 302.392,Z 451.465,A -85,B 0,C 180,E1 -16305.504,E2 -16305.504} C_VEL
LIN {X 0,Y 304.318,Z 443.736,A -85,B 0,C 180,E1 -16307.127,E2 -16307.127} C_VEL
LIN {X 0,Y 306.16,Z 436.315,A -85,B 0,C 180,E1 -16308.401,E2 -16308.401} C_VEL
LIN {X 0,Y 308.511,Z 426.101,A -85,B 0,C 180,E1 -16309.809,E2 -16309.809} C_VEL
LIN {X 0,Y 310.54,Z 415.838,A -85,B 0,C 180,E1 -16310.884,E2 -16310.884} C_VEL
LIN {X 0,Y 312.31,Z 405.63,A -85,B 0,C 180,E1 -16311.711,E2 -16311.711} C_VEL
LIN {X 0,Y 314.214,Z 392.445,A -85,B 0,C 180,E1 -16312.49,E2 -16312.49} C_VEL
LIN {X 0,Y 317.504,Z 354.849,A -85,B 0,C 180,E1 -16314.027,E2 -16314.027} C_VEL
LIN {X 0,Y 316.102,Z 342.03,A -85,B 0,C 180,E1 -16314.99,E2 -16314.99} C_VEL
LIN {X 0,Y 313.761,Z 329.104,A -85,B 0,C 180,E1 -16316.223,E2 -16316.223} C_VEL
LIN {X 0,Y 311.96,Z 321.534,A -85,B 0,C 180,E1 -16317.074,E2 -16317.074} C_VEL
LIN {X 0,Y 309.685,Z 316.733,A -85,B 0,C 180,E1 -16317.915,E2 -16317.915} C_VEL
LIN {X 0,Y 307.215,Z 311.943,A -85,B 0,C 180,E1 -16318.841,E2 -16318.841} C_VEL
LIN {X 0,Y 304.836,Z 307.14,A -85,B 0,C 180,E1 -16319.908,E2 -16319.908} C_VEL
LIN {X 0,Y 303.088,Z 301.161,A -85,B 0,C 180,E1 -16322.721,E2 -16322.721} C_VEL
LIN {X 0,Y 301.361,Z 295.939,A -85,B 0,C 180,E1 -16325.666,E2 -16325.666} C_VEL
LIN {X 0,Y 299.936,Z 292.082,A -85,B 0,C 180,E1 -16328.386,E2 -16328.386} C_VEL
LIN {X 0,Y 298.395,Z 288.128,A -85,B 0,C 180,E1 -16332.508,E2 -16332.508} C_VEL
LIN {X 0,Y 298.377,Z 288.131,A -85,B 0,C 180,E1 -16335.033,E2 -16335.033} C_VEL
LIN {X 0,Y 298.359,Z 288.132,A -85,B 0,C 180,E1 -16338.921,E2 -16338.921} C_VEL
LIN {X 0,Y 298.401,Z 288.182,A -85,B 0,C 180,E1 -16342.639,E2 -16342.639} C_VEL
LIN {X 0,Y 300.16,Z 292.186,A -85,B 0,C 180,E1 -16346.612,E2 -16346.612} C_VEL
LIN {X 0,Y 301.871,Z 296.383,A -85,B 0,C 180,E1 -16349.254,E2 -16349.254} C_VEL
LIN {X 0,Y 305.958,Z 302.089,A -85,B 0,C 180,E1 -16350.937,E2 -16350.937} C_VEL
LIN {X 0,Y 310.189,Z 308.353,A -85,B 0,C 180,E1 -16352.491,E2 -16352.491} C_VEL
LIN {X 0,Y 314.053,Z 314.951,A -85,B 0,C 180,E1 -16353.82,E2 -16353.82} C_VEL
LIN {X 0,Y 318.465,Z 323.465,A -85,B 0,C 180,E1 -16355.219,E2 -16355.219} C_VEL
LIN {X 0,Y 319.612,Z 326.119,A -85,B 0,C 180,E1 -16355.595,E2 -16355.595} C_VEL
LIN {X 0,Y 314.994,Z 376.211,A -85,B 0,C 180,E1 -16357.625,E2 -16357.625} C_VEL
LIN {X 0,Y 313.672,Z 387.233,A -85,B 0,C 180,E1 -16358.298,E2 -16358.298} C_VEL
LIN {X 0,Y 312.012,Z 398.15,A -85,B 0,C 180,E1 -16359.215,E2 -16359.215} C_VEL
LIN {X 0,Y 310.243,Z 408.249,A -85,B 0,C 180,E1 -16360.302,E2 -16360.302} C_VEL
LIN {X 0,Y 308.062,Z 418.309,A -85,B 0,C 180,E1 -16361.713,E2 -16361.713} C_VEL
LIN {X 0,Y 306.361,Z 425.516,A -85,B 0,C 180,E1 -16362.987,E2 -16362.987} C_VEL
LIN {X 0,Y 304.816,Z 431.513,A -85,B 0,C 180,E1 -16364.275,E2 -16364.275} C_VEL
LIN {X 0,Y 303.359,Z 436.614,A -85,B 0,C 180,E1 -16365.573,E2 -16365.573} C_VEL
LIN {X 0,Y 301.774,Z 441.813,A -85,B 0,C 180,E1 -16367.212,E2 -16367.212} C_VEL
LIN {X 0,Y 300.597,Z 445.148,A -85,B 0,C 180,E1 -16368.531,E2 -16368.531} C_VEL
LIN {X 0,Y 299.524,Z 448.441,A -85,B 0,C 180,E1 -16370.234,E2 -16370.234} C_VEL
LIN {X 0,Y 298.494,Z 450.735,A -85,B 0,C 180,E1 -16371.872,E2 -16371.872} C_VEL
LIN {X 0,Y 297.812,Z 452.003,A -85,B 0,C 180,E1 -16373.217,E2 -16373.217} C_VEL
LIN {X 0,Y 297.432,Z 452.752,A -85,B 0,C 180,E1 -16374.57,E2 -16374.57} C_VEL
LIN {X 0,Y 297.113,Z 452.954,A -85,B 0,C 180,E1 -16375.924,E2 -16375.924} C_VEL
LIN {X 0,Y 296.821,Z 452.549,A -85,B 0,C 180,E1 -16377.279,E2 -16377.279} C_VEL
LIN {X 0,Y 296.629,Z 451.633,A -85,B 0,C 180,E1 -16378.636,E2 -16378.636} C_VEL
LIN {X 0,Y 296.562,Z 450.207,A -85,B 0,C 180,E1 -16379.993,E2 -16379.993} C_VEL
LIN {X 0,Y 296.577,Z 446.964,A -85,B 0,C 180,E1 -16382.03,E2 -16382.03} C_VEL
LIN {X 0,Y 296.735,Z 444.03,A -85,B 0,C 180,E1 -16383.388,E2 -16383.388} C_VEL
LIN {X 0,Y 296.79,Z 439.373,A -85,B 0,C 180,E1 -16385.087,E2 -16385.087} C_VEL
LIN {X 0,Y 297.062,Z 433.516,A -85,B 0,C 180,E1 -16386.786,E2 -16386.786} C_VEL
LIN {X 0,Y 297.46,Z 426.167,A -85,B 0,C 180,E1 -16388.484,E2 -16388.484} C_VEL
LIN {X 0,Y 297.896,Z 417.777,A -85,B 0,C 180,E1 -16390.013,E2 -16390.013} C_VEL
LIN {X 0,Y 298.218,Z 411.073,A -85,B 0,C 180,E1 -16391.032,E2 -16391.032} C_VEL
LIN {X 0,Y 298.674,Z 403.098,A -85,B 0,C 180,E1 -16392.046,E2 -16392.046} C_VEL
LIN {X 0,Y 299.08,Z 393.213,A -85,B 0,C 180,E1 -16393.064,E2 -16393.064} C_VEL
LIN {X 0,Y 299.619,Z 381.328,A -85,B 0,C 180,E1 -16393.991,E2 -16393.991} C_VEL
LIN {X 0,Y 299.93,Z 370.363,A -85,B 0,C 180,E1 -16394.582,E2 -16394.582} C_VEL
LIN {X 0,Y 301.165,Z 314.508,A -85,B 0,C 180,E1 -16396.613,E2 -16396.613} C_VEL
LIN {X 0,Y 298.68,Z 293.688,A -85,B 0,C 180,E1 -16397.428,E2 -16397.428} C_VEL
LIN {X 0,Y 298.618,Z 293.025,A -85,B 0,C 180,E1 -16397.453,E2 -16397.453} C_VEL
LIN {X 0,Y 298.652,Z 288.094,A -85,B 0,C 180,E1 -16399.306,E2 -16399.306} C_VEL
LIN {X 0,Y 298.377,Z 288.127,A -85,B 0,C 180,E1 -16403.596,E2 -16403.596} C_VEL
LIN {X 0,Y 298.388,Z 288.128,A -85,B 0,C 180,E1 -16406.575,E2 -16406.575} C_VEL
LIN {X 0,Y 298.341,Z 288.132,A -85,B 0,C 180,E1 -16409.64,E2 -16409.64} C_VEL
LIN {X 0,Y 298.374,Z 288.129,A -85,B 0,C 180,E1 -16412.793,E2 -16412.793} C_VEL
LIN {X 0,Y 298.406,Z 288.126,A -85,B 0,C 180,E1 -16416.794,E2 -16416.794} C_VEL
LIN {X 0,Y 298.322,Z 288.134,A -85,B 0,C 180,E1 -16421.26,E2 -16421.26} C_VEL
LIN {X 0,Y 298.327,Z 288.136,A -85,B 0,C 180,E1 -16425.027,E2 -16425.027} C_VEL
LIN {X 0,Y 298.347,Z 288.135,A -85,B 0,C 180,E1 -16428.73,E2 -16428.73} C_VEL
LIN {X 0,Y 298.373,Z 288.128,A -85,B 0,C 180,E1 -16432.233,E2 -16432.233} C_VEL
LIN {X 0,Y 298.371,Z 288.129,A -85,B 0,C 180,E1 -16435.574,E2 -16435.574} C_VEL
LIN {X 0,Y 298.344,Z 288.133,A -85,B 0,C 180,E1 -16438.783,E2 -16438.783} C_VEL
LIN {X 0,Y 298.404,Z 288.124,A -85,B 0,C 180,E1 -16441.896,E2 -16441.896} C_VEL
LIN {X 0,Y 298.438,Z 288.122,A -85,B 0,C 180,E1 -16444.918,E2 -16444.918} C_VEL
LIN {X 0,Y 298.391,Z 288.129,A -85,B 0,C 180,E1 -16449.309,E2 -16449.309} C_VEL
LIN {X 0,Y 298.487,Z 288.114,A -85,B 0,C 180,E1 -16452.174,E2 -16452.174} C_VEL
LIN {X 0,Y 298.539,Z 288.107,A -85,B 0,C 180,E1 -16454.99,E2 -16454.99} C_VEL
LIN {X 0,Y 298.545,Z 288.107,A -85,B 0,C 180,E1 -16459.143,E2 -16459.143} C_VEL
LIN {X 0,Y 298.701,Z 288.091,A -85,B 0,C 180,E1 -16461.882,E2 -16461.882} C_VEL
LIN {X 0,Y 298.611,Z 288.098,A -85,B 0,C 180,E1 -16464.596,E2 -16464.596} C_VEL
LIN {X 0,Y 298.877,Z 288.065,A -85,B 0,C 180,E1 -16468.65,E2 -16468.65} C_VEL
LIN {X 0,Y 298.876,Z 288.065,A -85,B 0,C 180,E1 -16471.345,E2 -16471.345} C_VEL
LIN {X 0,Y 298.607,Z 288.098,A -85,B 0,C 180,E1 -16475.4,E2 -16475.4} C_VEL
LIN {X 0,Y 298.697,Z 288.092,A -85,B 0,C 180,E1 -16478.113,E2 -16478.113} C_VEL
LIN {X 0,Y 298.501,Z 288.116,A -85,B 0,C 180,E1 -16482.231,E2 -16482.231} C_VEL
LIN {X 0,Y 298.511,Z 288.11,A -85,B 0,C 180,E1 -16485.179,E2 -16485.179} C_VEL
LIN {X 0,Y 298.471,Z 288.116,A -85,B 0,C 180,E1 -16489.245,E2 -16489.245} C_VEL
LIN {X 0,Y 298.377,Z 288.126,A -85,B 0,C 180,E1 -16493.602,E2 -16493.602} C_VEL
LIN {X 0,Y 298.434,Z 288.124,A -85,B 0,C 180,E1 -16496.577,E2 -16496.577} C_VEL
LIN {X 0,Y 298.37,Z 288.128,A -85,B 0,C 180,E1 -16499.643,E2 -16499.643} C_VEL
LIN {X 0,Y 298.345,Z 288.135,A -85,B 0,C 180,E1 -16502.803,E2 -16502.803} C_VEL
LIN {X 0,Y 298.417,Z 288.126,A -85,B 0,C 180,E1 -16506.816,E2 -16506.816} C_VEL
LIN {X 0,Y 298.408,Z 288.128,A -85,B 0,C 180,E1 -16511.254,E2 -16511.254} C_VEL
LIN {X 0,Y 298.445,Z 288.122,A -85,B 0,C 180,E1 -16515.065,E2 -16515.065} C_VEL
LIN {X 0,Y 298.411,Z 288.124,A -85,B 0,C 180,E1 -16518.903,E2 -16518.903} C_VEL
LIN {X 0,Y 298.425,Z 288.124,A -85,B 0,C 180,E1 -16523.193,E2 -16523.193} C_VEL
LIN {X 0,Y 298.357,Z 288.131,A -85,B 0,C 180,E1 -16527.205,E2 -16527.205} C_VEL
LIN {X 0,Y 298.391,Z 288.125,A -85,B 0,C 180,E1 -16530.622,E2 -16530.622} C_VEL
LIN {X 0,Y 298.449,Z 288.121,A -85,B 0,C 180,E1 -16533.481,E2 -16533.481} C_VEL
LIN {X 0,Y 298.4,Z 288.124,A -85,B 0,C 180,E1 -16536.706,E2 -16536.706} C_VEL
LIN {X 0,Y 298.449,Z 288.118,A -85,B 0,C 180,E1 -16540.759,E2 -16540.759} C_VEL
LIN {X 0,Y 298.56,Z 288.104,A -85,B 0,C 180,E1 -16545.001,E2 -16545.001} C_VEL
LIN {X 0,Y 298.555,Z 288.104,A -85,B 0,C 180,E1 -16549.338,E2 -16549.338} C_VEL
LIN {X 0,Y 298.696,Z 288.09,A -85,B 0,C 180,E1 -16551.892,E2 -16551.892} C_VEL
LIN {X 0,Y 298.619,Z 288.099,A -85,B 0,C 180,E1 -16554.605,E2 -16554.605} C_VEL
LIN {X 0,Y 298.568,Z 288.102,A -85,B 0,C 180,E1 -16555.202,E2 -16555.202} C_VEL
LIN {X 0,Y 297.884,Z 288.193,A -85,B 0,C 180,E1 -16556.33,E2 -16556.33} C_VEL
LIN {X 0,Y 295.126,Z 288.535,A -85,B 0,C 180,E1 -16558.172,E2 -16558.172} C_VEL
LIN {X 0,Y 292.84,Z 288.817,A -85,B 0,C 180,E1 -16559.665,E2 -16559.665} C_VEL
LIN {X 0,Y 291.903,Z 288.936,A -85,B 0,C 180,E1 -16560.819,E2 -16560.819} C_VEL
LIN {X 0,Y 291.847,Z 288.94,A -85,B 0,C 180,E1 -16561.209,E2 -16561.209} C_VEL
LIN {X 0,Y 291.59,Z 288.972,A -85,B 0,C 180,E1 -16565.539,E2 -16565.539} C_VEL
LIN {X 0,Y 291.656,Z 288.968,A -85,B 0,C 180,E1 -16568.916,E2 -16568.916} C_VEL
LIN {X 0,Y 291.498,Z 288.986,A -85,B 0,C 180,E1 -16572.539,E2 -16572.539} C_VEL
LIN {X 0,Y 291.453,Z 288.991,A -85,B 0,C 180,E1 -16575.388,E2 -16575.388} C_VEL
LIN {X 0,Y 291.386,Z 288.998,A -85,B 0,C 180,E1 -16579.848,E2 -16579.848} C_VEL
LIN {X 0,Y 291.323,Z 289.005,A -85,B 0,C 180,E1 -16584.218,E2 -16584.218} C_VEL
LIN {X 0,Y 291.349,Z 289.008,A -85,B 0,C 180,E1 -16587.285,E2 -16587.285} C_VEL
LIN {X 0,Y 291.318,Z 289.006,A -85,B 0,C 180,E1 -16590.445,E2 -16590.445} C_VEL
LIN {X 0,Y 291.344,Z 289.006,A -85,B 0,C 180,E1 -16593.705,E2 -16593.705} C_VEL
LIN {X 0,Y 291.349,Z 289.005,A -85,B 0,C 180,E1 -16597.252,E2 -16597.252} C_VEL
LIN {X 0,Y 291.302,Z 289.007,A -85,B 0,C 180,E1 -16600.654,E2 -16600.654} C_VEL
LIN {X 0,Y 291.286,Z 289.011,A -85,B 0,C 180,E1 -16604.409,E2 -16604.409} C_VEL
LIN {X 0,Y 291.299,Z 289.009,A -85,B 0,C 180,E1 -16608.417,E2 -16608.417} C_VEL
LIN {X 0,Y 291.339,Z 289.004,A -85,B 0,C 180,E1 -16611.16,E2 -16611.16} C_VEL
LIN {X 0,Y 291.362,Z 289.002,A -85,B 0,C 180,E1 -16614.63,E2 -16614.63} C_VEL
LIN {X 0,Y 291.373,Z 289.003,A -85,B 0,C 180,E1 -16617.954,E2 -16617.954} C_VEL
LIN {X 0,Y 291.441,Z 288.993,A -85,B 0,C 180,E1 -16622.733,E2 -16622.733} C_VEL
LIN {X 0,Y 291.53,Z 289.095,A -85,B 0,C 180,E1 -16623.642,E2 -16623.642} C_VEL
LIN {X 0,Y 292.873,Z 296.819,A -85,B 0,C 180,E1 -16626.303,E2 -16626.303} C_VEL
LIN {X 0,Y 292.3,Z 304.482,A -85,B 0,C 180,E1 -16628.862,E2 -16628.862} C_VEL
LIN {X 0,Y 291.227,Z 315.015,A -85,B 0,C 180,E1 -16632.355,E2 -16632.355} C_VEL
LIN {X 0,Y 292.266,Z 332.849,A -85,B 0,C 180,E1 -16633.051,E2 -16633.051} C_VEL
LIN {X 0,Y 293.769,Z 349.43,A -85,B 0,C 180,E1 -16633.7,E2 -16633.7} C_VEL
LIN {X 0,Y 292.73,Z 394.446,A -85,B 0,C 180,E1 -16635.446,E2 -16635.446} C_VEL
LIN {X 0,Y 292.298,Z 406.373,A -85,B 0,C 180,E1 -16636.179,E2 -16636.179} C_VEL
LIN {X 0,Y 291.746,Z 417.306,A -85,B 0,C 180,E1 -16637.127,E2 -16637.127} C_VEL
LIN {X 0,Y 291.128,Z 428.076,A -85,B 0,C 180,E1 -16638.338,E2 -16638.338} C_VEL
LIN {X 0,Y 290.7,Z 437.557,A -85,B 0,C 180,E1 -16639.732,E2 -16639.732} C_VEL
LIN {X 0,Y 290.376,Z 444.37,A -85,B 0,C 180,E1 -16640.951,E2 -16640.951} C_VEL
LIN {X 0,Y 290.131,Z 450.861,A -85,B 0,C 180,E1 -16642.346,E2 -16642.346} C_VEL
LIN {X 0,Y 289.957,Z 456.769,A -85,B 0,C 180,E1 -16643.891,E2 -16643.891} C_VEL
LIN {X 0,Y 289.847,Z 460.695,A -85,B 0,C 180,E1 -16645.134,E2 -16645.134} C_VEL
LIN {X 0,Y 289.71,Z 464.342,A -85,B 0,C 180,E1 -16646.525,E2 -16646.525} C_VEL
LIN {X 0,Y 289.761,Z 468.486,A -85,B 0,C 180,E1 -16648.613,E2 -16648.613} C_VEL
LIN {X 0,Y 289.849,Z 470.436,A -85,B 0,C 180,E1 -16650.002,E2 -16650.002} C_VEL
LIN {X 0,Y 289.465,Z 471.791,A -85,B 0,C 180,E1 -16651.394,E2 -16651.394} C_VEL
LIN {X 0,Y 289.485,Z 472.647,A -85,B 0,C 180,E1 -16652.785,E2 -16652.785} C_VEL
LIN {X 0,Y 289.516,Z 472.878,A -85,B 0,C 180,E1 -16654.179,E2 -16654.179} C_VEL
LIN {X 0,Y 289.578,Z 472.543,A -85,B 0,C 180,E1 -16655.66,E2 -16655.66} C_VEL
LIN {X 0,Y 289.807,Z 471.781,A -85,B 0,C 180,E1 -16656.967,E2 -16656.967} C_VEL
LIN {X 0,Y 290.195,Z 470.507,A -85,B 0,C 180,E1 -16658.357,E2 -16658.357} C_VEL
LIN {X 0,Y 291.138,Z 467.474,A -85,B 0,C 180,E1 -16660.433,E2 -16660.433} C_VEL
LIN {X 0,Y 292.521,Z 463.152,A -85,B 0,C 180,E1 -16662.49,E2 -16662.49} C_VEL
LIN {X 0,Y 293.988,Z 458.427,A -85,B 0,C 180,E1 -16664.186,E2 -16664.186} C_VEL
LIN {X 0,Y 296.058,Z 451.33,A -85,B 0,C 180,E1 -16666.198,E2 -16666.198} C_VEL
LIN {X 0,Y 298.155,Z 443.727,A -85,B 0,C 180,E1 -16667.846,E2 -16667.846} C_VEL
LIN {X 0,Y 300.374,Z 435.315,A -85,B 0,C 180,E1 -16669.301,E2 -16669.301} C_VEL
LIN {X 0,Y 302.887,Z 424.912,A -85,B 0,C 180,E1 -16670.725,E2 -16670.725} C_VEL
LIN {X 0,Y 305.128,Z 414.558,A -85,B 0,C 180,E1 -16671.804,E2 -16671.804} C_VEL
LIN {X 0,Y 307.005,Z 404.346,A -85,B 0,C 180,E1 -16672.638,E2 -16672.638} C_VEL
LIN {X 0,Y 308.943,Z 391.417,A -85,B 0,C 180,E1 -16673.393,E2 -16673.393} C_VEL
LIN {X 0,Y 312.221,Z 355.585,A -85,B 0,C 180,E1 -16674.909,E2 -16674.909} C_VEL
LIN {X 0,Y 310.984,Z 343.714,A -85,B 0,C 180,E1 -16675.869,E2 -16675.869} C_VEL
LIN {X 0,Y 308.703,Z 330.384,A -85,B 0,C 180,E1 -16677.207,E2 -16677.207} C_VEL
LIN {X 0,Y 307.49,Z 325.462,A -85,B 0,C 180,E1 -16677.821,E2 -16677.821} C_VEL
LIN {X 0,Y 304.156,Z 318.247,A -85,B 0,C 180,E1 -16679.168,E2 -16679.168} C_VEL
LIN {X 0,Y 300.834,Z 312.132,A -85,B 0,C 180,E1 -16680.574,E2 -16680.574} C_VEL
LIN {X 0,Y 297.609,Z 306.311,A -85,B 0,C 180,E1 -16682.18,E2 -16682.18} C_VEL
LIN {X 0,Y 295.802,Z 300.705,A -85,B 0,C 180,E1 -16685.383,E2 -16685.383} C_VEL
LIN {X 0,Y 294.521,Z 296.993,A -85,B 0,C 180,E1 -16688.044,E2 -16688.044} C_VEL
LIN {X 0,Y 293.031,Z 293.199,A -85,B 0,C 180,E1 -16691.963,E2 -16691.963} C_VEL
LIN {X 0,Y 292.397,Z 292.004,A -85,B 0,C 180,E1 -16694.192,E2 -16694.192} C_VEL
LIN {X 0,Y 292.061,Z 291.401,A -85,B 0,C 180,E1 -16697.634,E2 -16697.634} C_VEL
LIN {X 0,Y 292.673,Z 292.31,A -85,B 0,C 180,E1 -16701.36,E2 -16701.36} C_VEL
LIN {X 0,Y 293.243,Z 293.464,A -85,B 0,C 180,E1 -16703.184,E2 -16703.184} C_VEL
LIN {X 0,Y 294.943,Z 297.286,A -85,B 0,C 180,E1 -16706.807,E2 -16706.807} C_VEL
LIN {X 0,Y 298.353,Z 301.779,A -85,B 0,C 180,E1 -16708.566,E2 -16708.566} C_VEL
LIN {X 0,Y 302.57,Z 307.712,A -85,B 0,C 180,E1 -16710.438,E2 -16710.438} C_VEL
LIN {X 0,Y 307.56,Z 315.48,A -85,B 0,C 180,E1 -16712.37,E2 -16712.37} C_VEL
LIN {X 0,Y 311.425,Z 322.637,A -85,B 0,C 180,E1 -16713.759,E2 -16713.759} C_VEL
LIN {X 0,Y 314.431,Z 328.921,A -85,B 0,C 180,E1 -16714.768,E2 -16714.768} C_VEL
LIN {X 0,Y 309.581,Z 377.384,A -85,B 0,C 180,E1 -16716.807,E2 -16716.807} C_VEL
LIN {X 0,Y 308.096,Z 388.67,A -85,B 0,C 180,E1 -16717.531,E2 -16717.531} C_VEL
LIN {X 0,Y 306.627,Z 397.719,A -85,B 0,C 180,E1 -16718.304,E2 -16718.304} C_VEL
LIN {X 0,Y 304.953,Z 406.482,A -85,B 0,C 180,E1 -16719.241,E2 -16719.241} C_VEL
LIN {X 0,Y 302.895,Z 415.965,A -85,B 0,C 180,E1 -16720.51,E2 -16720.51} C_VEL
LIN {X 0,Y 300.689,Z 424.531,A -85,B 0,C 180,E1 -16721.953,E2 -16721.953} C_VEL
LIN {X 0,Y 299.02,Z 430.753,A -85,B 0,C 180,E1 -16723.261,E2 -16723.261} C_VEL
LIN {X 0,Y 297.038,Z 437.138,A -85,B 0,C 180,E1 -16724.908,E2 -16724.908} C_VEL
LIN {X 0,Y 295.622,Z 441.321,A -85,B 0,C 180,E1 -16726.241,E2 -16726.241} C_VEL
LIN {X 0,Y 293.742,Z 446.326,A -85,B 0,C 180,E1 -16728.26,E2 -16728.26} C_VEL
LIN {X 0,Y 292.457,Z 449.9,A -85,B 0,C 180,E1 -16730.309,E2 -16730.309} C_VEL
LIN {X 0,Y 291.524,Z 451.516,A -85,B 0,C 180,E1 -16731.677,E2 -16731.677} C_VEL
LIN {X 0,Y 290.81,Z 452.582,A -85,B 0,C 180,E1 -16733.053,E2 -16733.053} C_VEL
LIN {X 0,Y 290.391,Z 453.141,A -85,B 0,C 180,E1 -16734.438,E2 -16734.438} C_VEL
LIN {X 0,Y 290.051,Z 453.221,A -85,B 0,C 180,E1 -16735.825,E2 -16735.825} C_VEL
LIN {X 0,Y 289.748,Z 452.742,A -85,B 0,C 180,E1 -16737.213,E2 -16737.213} C_VEL
LIN {X 0,Y 289.549,Z 451.657,A -85,B 0,C 180,E1 -16738.602,E2 -16738.602} C_VEL
LIN {X 0,Y 289.452,Z 449.116,A -85,B 0,C 180,E1 -16740.689,E2 -16740.689} C_VEL
LIN {X 0,Y 289.581,Z 445.158,A -85,B 0,C 180,E1 -16742.775,E2 -16742.775} C_VEL
LIN {X 0,Y 289.73,Z 440.742,A -85,B 0,C 180,E1 -16744.514,E2 -16744.514} C_VEL
LIN {X 0,Y 289.835,Z 435.425,A -85,B 0,C 180,E1 -16746.17,E2 -16746.17} C_VEL
LIN {X 0,Y 290.181,Z 429.601,A -85,B 0,C 180,E1 -16747.647,E2 -16747.647} C_VEL
LIN {X 0,Y 290.492,Z 422.968,A -85,B 0,C 180,E1 -16749.04,E2 -16749.04} C_VEL
LIN {X 0,Y 290.874,Z 413.859,A -85,B 0,C 180,E1 -16750.609,E2 -16750.609} C_VEL
LIN {X 0,Y 291.563,Z 403.476,A -85,B 0,C 180,E1 -16751.992,E2 -16751.992} C_VEL
LIN {X 0,Y 291.978,Z 393.614,A -85,B 0,C 180,E1 -16753.034,E2 -16753.034} C_VEL
LIN {X 0,Y 292.544,Z 381.11,A -85,B 0,C 180,E1 -16754.026,E2 -16754.026} C_VEL
LIN {X 0,Y 292.801,Z 370.934,A -85,B 0,C 180,E1 -16754.59,E2 -16754.59} C_VEL
LIN {X 0,Y 294.1,Z 315.273,A -85,B 0,C 180,E1 -16756.714,E2 -16756.714} C_VEL
LIN {X 0,Y 291.57,Z 293.573,A -85,B 0,C 180,E1 -16757.579,E2 -16757.579} C_VEL
LIN {X 0,Y 291.571,Z 293.119,A -85,B 0,C 180,E1 -16757.654,E2 -16757.654} C_VEL
LIN {X 0,Y 291.626,Z 288.969,A -85,B 0,C 180,E1 -16759.252,E2 -16759.252} C_VEL
LIN {X 0,Y 291.322,Z 289.011,A -85,B 0,C 180,E1 -16764.203,E2 -16764.203} C_VEL
LIN {X 0,Y 291.314,Z 289.007,A -85,B 0,C 180,E1 -16767.273,E2 -16767.273} C_VEL
LIN {X 0,Y 291.285,Z 289.014,A -85,B 0,C 180,E1 -16770.433,E2 -16770.433} C_VEL
LIN {X 0,Y 291.325,Z 289.005,A -85,B 0,C 180,E1 -16773.69,E2 -16773.69} C_VEL
LIN {X 0,Y 291.333,Z 289.005,A -85,B 0,C 180,E1 -16777.24,E2 -16777.24} C_VEL
LIN {X 0,Y 291.269,Z 289.012,A -85,B 0,C 180,E1 -16781.58,E2 -16781.58} C_VEL
LIN {X 0,Y 291.262,Z 289.014,A -85,B 0,C 180,E1 -16785.59,E2 -16785.59} C_VEL
LIN {X 0,Y 291.298,Z 289.009,A -85,B 0,C 180,E1 -16789.349,E2 -16789.349} C_VEL
LIN {X 0,Y 291.369,Z 289.005,A -85,B 0,C 180,E1 -16792.912,E2 -16792.912} C_VEL
LIN {X 0,Y 291.307,Z 289.008,A -85,B 0,C 180,E1 -16796.294,E2 -16796.294} C_VEL
LIN {X 0,Y 291.339,Z 289.003,A -85,B 0,C 180,E1 -16800.257,E2 -16800.257} C_VEL
LIN {X 0,Y 291.368,Z 289,A -85,B 0,C 180,E1 -16804.265,E2 -16804.265} C_VEL
LIN {X 0,Y 291.331,Z 289.009,A -85,B 0,C 180,E1 -16807.293,E2 -16807.293} C_VEL
LIN {X 0,Y 291.414,Z 288.994,A -85,B 0,C 180,E1 -16810.265,E2 -16810.265} C_VEL
LIN {X 0,Y 291.47,Z 288.987,A -85,B 0,C 180,E1 -16814.647,E2 -16814.647} C_VEL
LIN {X 0,Y 291.488,Z 288.985,A -85,B 0,C 180,E1 -16818.877,E2 -16818.877} C_VEL
LIN {X 0,Y 291.653,Z 288.97,A -85,B 0,C 180,E1 -16821.685,E2 -16821.685} C_VEL
LIN {X 0,Y 291.581,Z 288.974,A -85,B 0,C 180,E1 -16824.465,E2 -16824.465} C_VEL
LIN {X 0,Y 291.843,Z 288.942,A -85,B 0,C 180,E1 -16828.618,E2 -16828.618} C_VEL
LIN {X 0,Y 291.843,Z 288.942,A -85,B 0,C 180,E1 -16831.378,E2 -16831.378} C_VEL
LIN {X 0,Y 291.577,Z 288.974,A -85,B 0,C 180,E1 -16835.53,E2 -16835.53} C_VEL
LIN {X 0,Y 291.649,Z 288.97,A -85,B 0,C 180,E1 -16838.311,E2 -16838.311} C_VEL
LIN {X 0,Y 291.467,Z 288.99,A -85,B 0,C 180,E1 -16842.531,E2 -16842.531} C_VEL
LIN {X 0,Y 291.458,Z 288.989,A -85,B 0,C 180,E1 -16845.379,E2 -16845.379} C_VEL
LIN {X 0,Y 291.399,Z 288.997,A -85,B 0,C 180,E1 -16849.876,E2 -16849.876} C_VEL
LIN {X 0,Y 291.33,Z 289.006,A -85,B 0,C 180,E1 -16854.209,E2 -16854.209} C_VEL
LIN {X 0,Y 291.369,Z 289.001,A -85,B 0,C 180,E1 -16857.274,E2 -16857.274} C_VEL
LIN {X 0,Y 291.286,Z 289.012,A -85,B 0,C 180,E1 -16860.439,E2 -16860.439} C_VEL
LIN {X 0,Y 291.295,Z 289.009,A -85,B 0,C 180,E1 -16863.702,E2 -16863.702} C_VEL
LIN {X 0,Y 291.351,Z 289.006,A -85,B 0,C 180,E1 -16867.263,E2 -16867.263} C_VEL
LIN {X 0,Y 291.355,Z 289.002,A -85,B 0,C 180,E1 -16870.635,E2 -16870.635} C_VEL
LIN {X 0,Y 291.362,Z 289.001,A -85,B 0,C 180,E1 -16874.384,E2 -16874.384} C_VEL
LIN {X 0,Y 291.346,Z 289.002,A -85,B 0,C 180,E1 -16878.396,E2 -16878.396} C_VEL
LIN {X 0,Y 291.338,Z 289.006,A -85,B 0,C 180,E1 -16881.167,E2 -16881.167} C_VEL
LIN {X 0,Y 291.346,Z 289.003,A -85,B 0,C 180,E1 -16884.635,E2 -16884.635} C_VEL
LIN {X 0,Y 291.333,Z 289.006,A -85,B 0,C 180,E1 -16887.956,E2 -16887.956} C_VEL
LIN {X 0,Y 291.342,Z 289.004,A -85,B 0,C 180,E1 -16891.164,E2 -16891.164} C_VEL
LIN {X 0,Y 291.382,Z 289,A -85,B 0,C 180,E1 -16894.278,E2 -16894.278} C_VEL
LIN {X 0,Y 291.341,Z 289.004,A -85,B 0,C 180,E1 -16897.305,E2 -16897.305} C_VEL
LIN {X 0,Y 291.377,Z 289.002,A -85,B 0,C 180,E1 -16900.273,E2 -16900.273} C_VEL
LIN {X 0,Y 291.472,Z 288.988,A -85,B 0,C 180,E1 -16904.672,E2 -16904.672} C_VEL
LIN {X 0,Y 291.505,Z 288.983,A -85,B 0,C 180,E1 -16908.887,E2 -16908.887} C_VEL
LIN {X 0,Y 291.646,Z 288.967,A -85,B 0,C 180,E1 -16911.694,E2 -16911.694} C_VEL
LIN {X 0,Y 291.589,Z 288.976,A -85,B 0,C 180,E1 -16914.475,E2 -16914.475} C_VEL
LIN {X 0,Y 291.865,Z 288.942,A -85,B 0,C 180,E1 -16918.627,E2 -16918.627} C_VEL
LIN {X 0,Y 291.847,Z 288.94,A -85,B 0,C 180,E1 -16921.209,E2 -16921.209} C_VEL
LIN {X 0,Y 291.224,Z 289.022,A -85,B 0,C 180,E1 -16922.358,E2 -16922.358} C_VEL
LIN {X 0,Y 288.34,Z 289.386,A -85,B 0,C 180,E1 -16924.226,E2 -16924.226} C_VEL
LIN {X 0,Y 285.834,Z 289.696,A -85,B 0,C 180,E1 -16925.742,E2 -16925.742} C_VEL
LIN {X 0,Y 284.722,Z 289.831,A -85,B 0,C 180,E1 -16926.919,E2 -16926.919} C_VEL
LIN {X 0,Y 284.614,Z 289.842,A -85,B 0,C 180,E1 -16927.319,E2 -16927.319} C_VEL
LIN {X 0,Y 284.503,Z 289.856,A -85,B 0,C 180,E1 -16929.964,E2 -16929.964} C_VEL
LIN {X 0,Y 284.41,Z 289.867,A -85,B 0,C 180,E1 -16934.313,E2 -16934.313} C_VEL
LIN {X 0,Y 284.315,Z 289.882,A -85,B 0,C 180,E1 -16938.751,E2 -16938.751} C_VEL
LIN {X 0,Y 284.293,Z 289.881,A -85,B 0,C 180,E1 -16941.772,E2 -16941.772} C_VEL
LIN {X 0,Y 284.28,Z 289.885,A -85,B 0,C 180,E1 -16944.858,E2 -16944.858} C_VEL
LIN {X 0,Y 284.28,Z 289.883,A -85,B 0,C 180,E1 -16948.022,E2 -16948.022} C_VEL
LIN {X 0,Y 284.285,Z 289.886,A -85,B 0,C 180,E1 -16951.282,E2 -16951.282} C_VEL
LIN {X 0,Y 284.337,Z 289.88,A -85,B 0,C 180,E1 -16955.352,E2 -16955.352} C_VEL
LIN {X 0,Y 284.295,Z 289.882,A -85,B 0,C 180,E1 -16958.178,E2 -16958.178} C_VEL
LIN {X 0,Y 284.239,Z 289.89,A -85,B 0,C 180,E1 -16962.122,E2 -16962.122} C_VEL
LIN {X 0,Y 284.242,Z 289.89,A -85,B 0,C 180,E1 -16966.191,E2 -16966.191} C_VEL
LIN {X 0,Y 284.291,Z 289.885,A -85,B 0,C 180,E1 -16970.035,E2 -16970.035} C_VEL
LIN {X 0,Y 284.324,Z 289.88,A -85,B 0,C 180,E1 -16973.616,E2 -16973.616} C_VEL
LIN {X 0,Y 284.315,Z 289.878,A -85,B 0,C 180,E1 -16977.196,E2 -16977.196} C_VEL
LIN {X 0,Y 284.319,Z 289.882,A -85,B 0,C 180,E1 -16980.375,E2 -16980.375} C_VEL
LIN {X 0,Y 284.483,Z 289.951,A -85,B 0,C 180,E1 -16983.65,E2 -16983.65} C_VEL
LIN {X 0,Y 285.792,Z 297.27,A -85,B 0,C 180,E1 -16986.237,E2 -16986.237} C_VEL
LIN {X 0,Y 285.229,Z 304.539,A -85,B 0,C 180,E1 -16988.729,E2 -16988.729} C_VEL
LIN {X 0,Y 284.162,Z 314.92,A -85,B 0,C 180,E1 -16992.227,E2 -16992.227} C_VEL
LIN {X 0,Y 285.123,Z 332.468,A -85,B 0,C 180,E1 -16992.943,E2 -16992.943} C_VEL
LIN {X 0,Y 286.632,Z 350.587,A -85,B 0,C 180,E1 -16993.678,E2 -16993.678} C_VEL
LIN {X 0,Y 285.637,Z 394.393,A -85,B 0,C 180,E1 -16995.441,E2 -16995.441} C_VEL
LIN {X 0,Y 285.219,Z 406.215,A -85,B 0,C 180,E1 -16996.192,E2 -16996.192} C_VEL
LIN {X 0,Y 284.669,Z 417.111,A -85,B 0,C 180,E1 -16997.165,E2 -16997.165} C_VEL
LIN {X 0,Y 284.041,Z 427.853,A -85,B 0,C 180,E1 -16998.405,E2 -16998.405} C_VEL
LIN {X 0,Y 283.619,Z 437.322,A -85,B 0,C 180,E1 -16999.833,E2 -16999.833} C_VEL
LIN {X 0,Y 283.297,Z 444.131,A -85,B 0,C 180,E1 -17001.083,E2 -17001.083} C_VEL
LIN {X 0,Y 283.071,Z 450.624,A -85,B 0,C 180,E1 -17002.513,E2 -17002.513} C_VEL
LIN {X 0,Y 282.916,Z 455.827,A -85,B 0,C 180,E1 -17003.9,E2 -17003.9} C_VEL
LIN {X 0,Y 282.811,Z 459.402,A -85,B 0,C 180,E1 -17005.013,E2 -17005.013} C_VEL
LIN {X 0,Y 282.693,Z 463.231,A -85,B 0,C 180,E1 -17006.439,E2 -17006.439} C_VEL
LIN {X 0,Y 282.72,Z 467.547,A -85,B 0,C 180,E1 -17008.578,E2 -17008.578} C_VEL
LIN {X 0,Y 282.789,Z 469.688,A -85,B 0,C 180,E1 -17010.002,E2 -17010.002} C_VEL
LIN {X 0,Y 282.39,Z 471.204,A -85,B 0,C 180,E1 -17011.428,E2 -17011.428} C_VEL
LIN {X 0,Y 282.415,Z 472.124,A -85,B 0,C 180,E1 -17012.855,E2 -17012.855} C_VEL
LIN {X 0,Y 282.441,Z 472.491,A -85,B 0,C 180,E1 -17014.283,E2 -17014.283} C_VEL
LIN {X 0,Y 282.503,Z 472.366,A -85,B 0,C 180,E1 -17015.713,E2 -17015.713} C_VEL
LIN {X 0,Y 282.764,Z 471.769,A -85,B 0,C 180,E1 -17017.141,E2 -17017.141} C_VEL
LIN {X 0,Y 283.176,Z 470.609,A -85,B 0,C 180,E1 -17018.566,E2 -17018.566} C_VEL
LIN {X 0,Y 284.183,Z 467.846,A -85,B 0,C 180,E1 -17020.691,E2 -17020.691} C_VEL
LIN {X 0,Y 285.622,Z 463.755,A -85,B 0,C 180,E1 -17022.797,E2 -17022.797} C_VEL
LIN {X 0,Y 287.51,Z 458.311,A -85,B 0,C 180,E1 -17024.875,E2 -17024.875} C_VEL
LIN {X 0,Y 289.337,Z 452.548,A -85,B 0,C 180,E1 -17026.585,E2 -17026.585} C_VEL
LIN {X 0,Y 291.544,Z 445.42,A -85,B 0,C 180,E1 -17028.265,E2 -17028.265} C_VEL
LIN {X 0,Y 294.138,Z 436.508,A -85,B 0,C 180,E1 -17029.908,E2 -17029.908} C_VEL
LIN {X 0,Y 296.453,Z 427.778,A -85,B 0,C 180,E1 -17031.196,E2 -17031.196} C_VEL
LIN {X 0,Y 299.112,Z 416.887,A -85,B 0,C 180,E1 -17032.448,E2 -17032.448} C_VEL
LIN {X 0,Y 301.221,Z 406.236,A -85,B 0,C 180,E1 -17033.37,E2 -17033.37} C_VEL
LIN {X 0,Y 303.244,Z 394.824,A -85,B 0,C 180,E1 -17034.111,E2 -17034.111} C_VEL
LIN {X 0,Y 305.107,Z 377.646,A -85,B 0,C 180,E1 -17034.918,E2 -17034.918} C_VEL
LIN {X 0,Y 307.177,Z 357.363,A -85,B 0,C 180,E1 -17035.769,E2 -17035.769} C_VEL
LIN {X 0,Y 306.106,Z 346.218,A -85,B 0,C 180,E1 -17036.708,E2 -17036.708} C_VEL
LIN {X 0,Y 304.158,Z 333.718,A -85,B 0,C 180,E1 -17038.019,E2 -17038.019} C_VEL
LIN {X 0,Y 303.175,Z 329.5,A -85,B 0,C 180,E1 -17038.563,E2 -17038.563} C_VEL
LIN {X 0,Y 299.646,Z 321.989,A -85,B 0,C 180,E1 -17040.108,E2 -17040.108} C_VEL
LIN {X 0,Y 297.448,Z 317.6,A -85,B 0,C 180,E1 -17041.159,E2 -17041.159} C_VEL
LIN {X 0,Y 294.056,Z 311.563,A -85,B 0,C 180,E1 -17042.907,E2 -17042.907} C_VEL
LIN {X 0,Y 290.201,Z 305.206,A -85,B 0,C 180,E1 -17045.277,E2 -17045.277} C_VEL
LIN {X 0,Y 289.256,Z 302.221,A -85,B 0,C 180,E1 -17047.406,E2 -17047.406} C_VEL
LIN {X 0,Y 288.434,Z 300.103,A -85,B 0,C 180,E1 -17049.312,E2 -17049.312} C_VEL
LIN {X 0,Y 287.437,Z 297.308,A -85,B 0,C 180,E1 -17052.811,E2 -17052.811} C_VEL
LIN {X 0,Y 286.889,Z 296.404,A -85,B 0,C 180,E1 -17055.272,E2 -17055.272} C_VEL
LIN {X 0,Y 286.831,Z 296.222,A -85,B 0,C 180,E1 -17058.574,E2 -17058.574} C_VEL
LIN {X 0,Y 287.779,Z 297.56,A -85,B 0,C 180,E1 -17062.365,E2 -17062.365} C_VEL
LIN {X 0,Y 288.147,Z 298.714,A -85,B 0,C 180,E1 -17063.601,E2 -17063.601} C_VEL
LIN {X 0,Y 292.447,Z 303.856,A -85,B 0,C 180,E1 -17066.491,E2 -17066.491} C_VEL
LIN {X 0,Y 296.404,Z 309.256,A -85,B 0,C 180,E1 -17068.607,E2 -17068.607} C_VEL
LIN {X 0,Y 299.458,Z 313.805,A -85,B 0,C 180,E1 -17070.037,E2 -17070.037} C_VEL
LIN {X 0,Y 303.889,Z 320.86,A -85,B 0,C 180,E1 -17071.851,E2 -17071.851} C_VEL
LIN {X 0,Y 308.181,Z 329.191,A -85,B 0,C 180,E1 -17073.476,E2 -17073.476} C_VEL
LIN {X 0,Y 309.324,Z 331.735,A -85,B 0,C 180,E1 -17073.908,E2 -17073.908} C_VEL
LIN {X 0,Y 304.431,Z 377.715,A -85,B 0,C 180,E1 -17075.894,E2 -17075.894} C_VEL
LIN {X 0,Y 302.919,Z 388.367,A -85,B 0,C 180,E1 -17076.584,E2 -17076.584} C_VEL
LIN {X 0,Y 301.042,Z 398.963,A -85,B 0,C 180,E1 -17077.519,E2 -17077.519} C_VEL
LIN {X 0,Y 298.987,Z 408.943,A -85,B 0,C 180,E1 -17078.627,E2 -17078.627} C_VEL
LIN {X 0,Y 296.794,Z 417.96,A -85,B 0,C 180,E1 -17079.912,E2 -17079.912} C_VEL
LIN {X 0,Y 294.708,Z 425.304,A -85,B 0,C 180,E1 -17081.214,E2 -17081.214} C_VEL
LIN {X 0,Y 292.879,Z 431.399,A -85,B 0,C 180,E1 -17082.539,E2 -17082.539} C_VEL
LIN {X 0,Y 290.788,Z 437.728,A -85,B 0,C 180,E1 -17084.216,E2 -17084.216} C_VEL
LIN {X 0,Y 288.898,Z 442.824,A -85,B 0,C 180,E1 -17085.914,E2 -17085.914} C_VEL
LIN {X 0,Y 286.907,Z 447.536,A -85,B 0,C 180,E1 -17087.976,E2 -17087.976} C_VEL
LIN {X 0,Y 285.512,Z 450.724,A -85,B 0,C 180,E1 -17090.071,E2 -17090.071} C_VEL
LIN {X 0,Y 284.56,Z 452.265,A -85,B 0,C 180,E1 -17091.471,E2 -17091.471} C_VEL
LIN {X 0,Y 283.811,Z 453.177,A -85,B 0,C 180,E1 -17092.881,E2 -17092.881} C_VEL
LIN {X 0,Y 283.354,Z 453.542,A -85,B 0,C 180,E1 -17094.299,E2 -17094.299} C_VEL
LIN {X 0,Y 282.993,Z 453.425,A -85,B 0,C 180,E1 -17095.72,E2 -17095.72} C_VEL
LIN {X 0,Y 282.677,Z 452.821,A -85,B 0,C 180,E1 -17097.143,E2 -17097.143} C_VEL
LIN {X 0,Y 282.47,Z 451.665,A -85,B 0,C 180,E1 -17098.567,E2 -17098.567} C_VEL
LIN {X 0,Y 282.372,Z 448.81,A -85,B 0,C 180,E1 -17100.706,E2 -17100.706} C_VEL
LIN {X 0,Y 282.431,Z 446.219,A -85,B 0,C 180,E1 -17102.132,E2 -17102.132} C_VEL
LIN {X 0,Y 282.663,Z 440.984,A -85,B 0,C 180,E1 -17104.27,E2 -17104.27} C_VEL
LIN {X 0,Y 282.762,Z 434.972,A -85,B 0,C 180,E1 -17106.164,E2 -17106.164} C_VEL
LIN {X 0,Y 283.133,Z 428.356,A -85,B 0,C 180,E1 -17107.839,E2 -17107.839} C_VEL
LIN {X 0,Y 283.598,Z 419.484,A -85,B 0,C 180,E1 -17109.622,E2 -17109.622} C_VEL
LIN {X 0,Y 283.936,Z 411.781,A -85,B 0,C 180,E1 -17110.871,E2 -17110.871} C_VEL
LIN {X 0,Y 284.456,Z 403.852,A -85,B 0,C 180,E1 -17111.934,E2 -17111.934} C_VEL
LIN {X 0,Y 284.872,Z 394.014,A -85,B 0,C 180,E1 -17113.002,E2 -17113.002} C_VEL
LIN {X 0,Y 285.401,Z 382.293,A -85,B 0,C 180,E1 -17113.975,E2 -17113.975} C_VEL
LIN {X 0,Y 285.707,Z 371.549,A -85,B 0,C 180,E1 -17114.596,E2 -17114.596} C_VEL
LIN {X 0,Y 286.926,Z 315.354,A -85,B 0,C 180,E1 -17116.815,E2 -17116.815} C_VEL
LIN {X 0,Y 284.496,Z 293.512,A -85,B 0,C 180,E1 -17117.746,E2 -17117.746} C_VEL
LIN {X 0,Y 284.588,Z 289.846,A -85,B 0,C 180,E1 -17119.185,E2 -17119.185} C_VEL
LIN {X 0,Y 284.287,Z 289.884,A -85,B 0,C 180,E1 -17123.834,E2 -17123.834} C_VEL
LIN {X 0,Y 284.272,Z 289.884,A -85,B 0,C 180,E1 -17127.121,E2 -17127.121} C_VEL
LIN {X 0,Y 284.257,Z 289.889,A -85,B 0,C 180,E1 -17130.075,E2 -17130.075} C_VEL
LIN {X 0,Y 284.287,Z 289.883,A -85,B 0,C 180,E1 -17132.937,E2 -17132.937} C_VEL
LIN {X 0,Y 284.298,Z 289.885,A -85,B 0,C 180,E1 -17136.38,E2 -17136.38} C_VEL
LIN {X 0,Y 284.231,Z 289.889,A -85,B 0,C 180,E1 -17139.995,E2 -17139.995} C_VEL
LIN {X 0,Y 284.206,Z 289.893,A -85,B 0,C 180,E1 -17144.18,E2 -17144.18} C_VEL
LIN {X 0,Y 284.228,Z 289.889,A -85,B 0,C 180,E1 -17148.114,E2 -17148.114} C_VEL
LIN {X 0,Y 284.274,Z 289.884,A -85,B 0,C 180,E1 -17151.823,E2 -17151.823} C_VEL
LIN {X 0,Y 284.273,Z 289.887,A -85,B 0,C 180,E1 -17155.343,E2 -17155.343} C_VEL
LIN {X 0,Y 284.25,Z 289.887,A -85,B 0,C 180,E1 -17158.718,E2 -17158.718} C_VEL
LIN {X 0,Y 284.351,Z 289.876,A -85,B 0,C 180,E1 -17162.823,E2 -17162.823} C_VEL
LIN {X 0,Y 284.29,Z 289.882,A -85,B 0,C 180,E1 -17166.698,E2 -17166.698} C_VEL
LIN {X 0,Y 284.353,Z 289.877,A -85,B 0,C 180,E1 -17171.256,E2 -17171.256} C_VEL
LIN {X 0,Y 284.423,Z 289.869,A -85,B 0,C 180,E1 -17175.692,E2 -17175.692} C_VEL
LIN {X 0,Y 284.518,Z 289.856,A -85,B 0,C 180,E1 -17180.041,E2 -17180.041} C_VEL
LIN {X 0,Y 284.642,Z 289.838,A -85,B 0,C 180,E1 -17182.906,E2 -17182.906} C_VEL
LIN {X 0,Y 284.707,Z 289.83,A -85,B 0,C 180,E1 -17187.168,E2 -17187.168} C_VEL
LIN {X 0,Y 284.884,Z 289.814,A -85,B 0,C 180,E1 -17189.998,E2 -17189.998} C_VEL
LIN {X 0,Y 284.706,Z 289.83,A -85,B 0,C 180,E1 -17192.827,E2 -17192.827} C_VEL
LIN {X 0,Y 284.638,Z 289.838,A -85,B 0,C 180,E1 -17197.089,E2 -17197.089} C_VEL
LIN {X 0,Y 284.514,Z 289.857,A -85,B 0,C 180,E1 -17199.955,E2 -17199.955} C_VEL
LIN {X 0,Y 284.417,Z 289.869,A -85,B 0,C 180,E1 -17204.303,E2 -17204.303} C_VEL
LIN {X 0,Y 284.346,Z 289.878,A -85,B 0,C 180,E1 -17208.74,E2 -17208.74} C_VEL
LIN {X 0,Y 284.281,Z 289.883,A -85,B 0,C 180,E1 -17213.297,E2 -17213.297} C_VEL
LIN {X 0,Y 284.344,Z 289.877,A -85,B 0,C 180,E1 -17217.175,E2 -17217.175} C_VEL
LIN {X 0,Y 284.245,Z 289.888,A -85,B 0,C 180,E1 -17221.277,E2 -17221.277} C_VEL
LIN {X 0,Y 284.313,Z 289.881,A -85,B 0,C 180,E1 -17225.357,E2 -17225.357} C_VEL
LIN {X 0,Y 284.284,Z 289.882,A -85,B 0,C 180,E1 -17228.17,E2 -17228.17} C_VEL
LIN {X 0,Y 284.297,Z 289.88,A -85,B 0,C 180,E1 -17232.145,E2 -17232.145} C_VEL
LIN {X 0,Y 284.309,Z 289.879,A -85,B 0,C 180,E1 -17236.213,E2 -17236.213} C_VEL
LIN {X 0,Y 284.311,Z 289.879,A -85,B 0,C 180,E1 -17240.018,E2 -17240.018} C_VEL
LIN {X 0,Y 284.312,Z 289.883,A -85,B 0,C 180,E1 -17243.622,E2 -17243.622} C_VEL
LIN {X 0,Y 284.27,Z 289.886,A -85,B 0,C 180,E1 -17247.196,E2 -17247.196} C_VEL
LIN {X 0,Y 284.32,Z 289.878,A -85,B 0,C 180,E1 -17250.382,E2 -17250.382} C_VEL
LIN {X 0,Y 284.344,Z 289.879,A -85,B 0,C 180,E1 -17253.593,E2 -17253.593} C_VEL
LIN {X 0,Y 284.302,Z 289.879,A -85,B 0,C 180,E1 -17256.711,E2 -17256.711} C_VEL
LIN {X 0,Y 284.348,Z 289.879,A -85,B 0,C 180,E1 -17259.911,E2 -17259.911} C_VEL
LIN {X 0,Y 284.422,Z 289.867,A -85,B 0,C 180,E1 -17264.499,E2 -17264.499} C_VEL
LIN {X 0,Y 284.458,Z 289.863,A -85,B 0,C 180,E1 -17268.608,E2 -17268.608} C_VEL
LIN {X 0,Y 284.6,Z 289.844,A -85,B 0,C 180,E1 -17271.487,E2 -17271.487} C_VEL
LIN {X 0,Y 284.559,Z 289.853,A -85,B 0,C 180,E1 -17274.338,E2 -17274.338} C_VEL
LIN {X 0,Y 284.831,Z 289.819,A -85,B 0,C 180,E1 -17278.593,E2 -17278.593} C_VEL
LIN {X 0,Y 284.826,Z 289.815,A -85,B 0,C 180,E1 -17281.421,E2 -17281.421} C_VEL
LIN {X 0,Y 284.63,Z 289.841,A -85,B 0,C 180,E1 -17287.098,E2 -17287.098} C_VEL
LIN {X 0,Y 284.614,Z 289.842,A -85,B 0,C 180,E1 -17287.319,E2 -17287.319} C_VEL
LIN {X 0,Y 283.889,Z 289.935,A -85,B 0,C 180,E1 -17288.498,E2 -17288.498} C_VEL
LIN {X 0,Y 280.976,Z 290.297,A -85,B 0,C 180,E1 -17290.418,E2 -17290.418} C_VEL
LIN {X 0,Y 278.52,Z 290.603,A -85,B 0,C 180,E1 -17291.977,E2 -17291.977} C_VEL
LIN {X 0,Y 277.452,Z 290.735,A -85,B 0,C 180,E1 -17293.187,E2 -17293.187} C_VEL
LIN {X 0,Y 277.356,Z 290.745,A -85,B 0,C 180,E1 -17293.597,E2 -17293.597} C_VEL
LIN {X 0,Y 277.334,Z 290.748,A -85,B 0,C 180,E1 -17296.193,E2 -17296.193} C_VEL
LIN {X 0,Y 277.256,Z 290.761,A -85,B 0,C 180,E1 -17300.793,E2 -17300.793} C_VEL
LIN {X 0,Y 277.233,Z 290.76,A -85,B 0,C 180,E1 -17304.138,E2 -17304.138} C_VEL
LIN {X 0,Y 277.266,Z 290.76,A -85,B 0,C 180,E1 -17307.488,E2 -17307.488} C_VEL
LIN {X 0,Y 277.248,Z 290.758,A -85,B 0,C 180,E1 -17310.479,E2 -17310.479} C_VEL
LIN {X 0,Y 277.247,Z 290.761,A -85,B 0,C 180,E1 -17313.902,E2 -17313.902} C_VEL
LIN {X 0,Y 277.25,Z 290.764,A -85,B 0,C 180,E1 -17317.479,E2 -17317.479} C_VEL
LIN {X 0,Y 277.187,Z 290.767,A -85,B 0,C 180,E1 -17321.247,E2 -17321.247} C_VEL
LIN {X 0,Y 277.179,Z 290.769,A -85,B 0,C 180,E1 -17325.238,E2 -17325.238} C_VEL
LIN {X 0,Y 277.19,Z 290.765,A -85,B 0,C 180,E1 -17328.764,E2 -17328.764} C_VEL
LIN {X 0,Y 277.255,Z 290.759,A -85,B 0,C 180,E1 -17332.532,E2 -17332.532} C_VEL
LIN {X 0,Y 277.255,Z 290.763,A -85,B 0,C 180,E1 -17336.109,E2 -17336.109} C_VEL
LIN {X 0,Y 277.239,Z 290.76,A -85,B 0,C 180,E1 -17339.539,E2 -17339.539} C_VEL
LIN {X 0,Y 277.443,Z 290.838,A -85,B 0,C 180,E1 -17343.689,E2 -17343.689} C_VEL
LIN {X 0,Y 278.701,Z 297.791,A -85,B 0,C 180,E1 -17346.208,E2 -17346.208} C_VEL
LIN {X 0,Y 278.197,Z 304.331,A -85,B 0,C 180,E1 -17348.515,E2 -17348.515} C_VEL
LIN {X 0,Y 277.098,Z 314.544,A -85,B 0,C 180,E1 -17352.093,E2 -17352.093} C_VEL
LIN {X 0,Y 277.936,Z 331.927,A -85,B 0,C 180,E1 -17352.833,E2 -17352.833} C_VEL
LIN {X 0,Y 279.585,Z 350.061,A -85,B 0,C 180,E1 -17353.589,E2 -17353.589} C_VEL
LIN {X 0,Y 278.518,Z 393.351,A -85,B 0,C 180,E1 -17355.387,E2 -17355.387} C_VEL
LIN {X 0,Y 278.123,Z 406.042,A -85,B 0,C 180,E1 -17356.206,E2 -17356.206} C_VEL
LIN {X 0,Y 277.594,Z 416.862,A -85,B 0,C 180,E1 -17357.204,E2 -17357.204} C_VEL
LIN {X 0,Y 276.956,Z 427.513,A -85,B 0,C 180,E1 -17358.475,E2 -17358.475} C_VEL
LIN {X 0,Y 276.557,Z 436.952,A -85,B 0,C 180,E1 -17359.941,E2 -17359.941} C_VEL
LIN {X 0,Y 276.251,Z 443.736,A -85,B 0,C 180,E1 -17361.222,E2 -17361.222} C_VEL
LIN {X 0,Y 276.04,Z 450.208,A -85,B 0,C 180,E1 -17362.689,E2 -17362.689} C_VEL
LIN {X 0,Y 275.863,Z 455.565,A -85,B 0,C 180,E1 -17364.154,E2 -17364.154} C_VEL
LIN {X 0,Y 275.726,Z 459.997,A -85,B 0,C 180,E1 -17365.617,E2 -17365.617} C_VEL
LIN {X 0,Y 275.625,Z 463.641,A -85,B 0,C 180,E1 -17367.079,E2 -17367.079} C_VEL
LIN {X 0,Y 275.678,Z 466.607,A -85,B 0,C 180,E1 -17368.542,E2 -17368.542} C_VEL
LIN {X 0,Y 275.73,Z 468.913,A -85,B 0,C 180,E1 -17370.002,E2 -17370.002} C_VEL
LIN {X 0,Y 275.328,Z 470.484,A -85,B 0,C 180,E1 -17371.465,E2 -17371.465} C_VEL
LIN {X 0,Y 275.347,Z 471.537,A -85,B 0,C 180,E1 -17372.929,E2 -17372.929} C_VEL
LIN {X 0,Y 275.393,Z 472.219,A -85,B 0,C 180,E1 -17375.529,E2 -17375.529} C_VEL
LIN {X 0,Y 275.72,Z 471.674,A -85,B 0,C 180,E1 -17377.325,E2 -17377.325} C_VEL
LIN {X 0,Y 276.15,Z 470.604,A -85,B 0,C 180,E1 -17378.786,E2 -17378.786} C_VEL
LIN {X 0,Y 277.209,Z 468.147,A -85,B 0,C 180,E1 -17380.964,E2 -17380.964} C_VEL
LIN {X 0,Y 278.74,Z 464.426,A -85,B 0,C 180,E1 -17383.118,E2 -17383.118} C_VEL
LIN {X 0,Y 280.726,Z 459.219,A -85,B 0,C 180,E1 -17385.243,E2 -17385.243} C_VEL
LIN {X 0,Y 282.636,Z 453.76,A -85,B 0,C 180,E1 -17386.99,E2 -17386.99} C_VEL
LIN {X 0,Y 284.946,Z 447.065,A -85,B 0,C 180,E1 -17388.704,E2 -17388.704} C_VEL
LIN {X 0,Y 287.675,Z 438.793,A -85,B 0,C 180,E1 -17390.375,E2 -17390.375} C_VEL
LIN {X 0,Y 290.389,Z 429.354,A -85,B 0,C 180,E1 -17391.848,E2 -17391.848} C_VEL
LIN {X 0,Y 292.739,Z 420.524,A -85,B 0,C 180,E1 -17392.965,E2 -17392.965} C_VEL
LIN {X 0,Y 295.396,Z 409.528,A -85,B 0,C 180,E1 -17394.046,E2 -17394.046} C_VEL
LIN {X 0,Y 297.603,Z 397.941,A -85,B 0,C 180,E1 -17394.878,E2 -17394.878} C_VEL
LIN {X 0,Y 299.295,Z 385.976,A -85,B 0,C 180,E1 -17395.517,E2 -17395.517} C_VEL
LIN {X 0,Y 302.26,Z 358.651,A -85,B 0,C 180,E1 -17396.711,E2 -17396.711} C_VEL
LIN {X 0,Y 301.268,Z 347.589,A -85,B 0,C 180,E1 -17397.71,E2 -17397.71} C_VEL
LIN {X 0,Y 299.446,Z 334.981,A -85,B 0,C 180,E1 -17399.121,E2 -17399.121} C_VEL
LIN {X 0,Y 296.322,Z 327.736,A -85,B 0,C 180,E1 -17400.606,E2 -17400.606} C_VEL
LIN {X 0,Y 294.13,Z 323.156,A -85,B 0,C 180,E1 -17401.733,E2 -17401.733} C_VEL
LIN {X 0,Y 291.222,Z 317.656,A -85,B 0,C 180,E1 -17403.361,E2 -17403.361} C_VEL
LIN {X 0,Y 287.319,Z 311.035,A -85,B 0,C 180,E1 -17405.951,E2 -17405.951} C_VEL
LIN {X 0,Y 283.914,Z 305.835,A -85,B 0,C 180,E1 -17408.972,E2 -17408.972} C_VEL
LIN {X 0,Y 282.369,Z 302.985,A -85,B 0,C 180,E1 -17411.27,E2 -17411.27} C_VEL
LIN {X 0,Y 281.712,Z 301.377,A -85,B 0,C 180,E1 -17414.312,E2 -17414.312} C_VEL
LIN {X 0,Y 281.615,Z 301.001,A -85,B 0,C 180,E1 -17417.631,E2 -17417.631} C_VEL
LIN {X 0,Y 283.46,Z 302.839,A -85,B 0,C 180,E1 -17420.82,E2 -17420.82} C_VEL
LIN {X 0,Y 285.733,Z 304.934,A -85,B 0,C 180,E1 -17423.057,E2 -17423.057} C_VEL
LIN {X 0,Y 289.822,Z 310.148,A -85,B 0,C 180,E1 -17426.094,E2 -17426.094} C_VEL
LIN {X 0,Y 293.575,Z 315.507,A -85,B 0,C 180,E1 -17428.235,E2 -17428.235} C_VEL
LIN {X 0,Y 296.43,Z 319.848,A -85,B 0,C 180,E1 -17429.613,E2 -17429.613} C_VEL
LIN {X 0,Y 300.31,Z 326.281,A -85,B 0,C 180,E1 -17431.311,E2 -17431.311} C_VEL
LIN {X 0,Y 304.294,Z 334.364,A -85,B 0,C 180,E1 -17432.94,E2 -17432.94} C_VEL
LIN {X 0,Y 304.429,Z 335.605,A -85,B 0,C 180,E1 -17433.059,E2 -17433.059} C_VEL
LIN {X 0,Y 299.393,Z 378.434,A -85,B 0,C 180,E1 -17434.96,E2 -17434.96} C_VEL
LIN {X 0,Y 297.553,Z 390.326,A -85,B 0,C 180,E1 -17435.765,E2 -17435.765} C_VEL
LIN {X 0,Y 295.879,Z 399.093,A -85,B 0,C 180,E1 -17436.549,E2 -17436.549} C_VEL
LIN {X 0,Y 293.67,Z 408.96,A -85,B 0,C 180,E1 -17437.666,E2 -17437.666} C_VEL
LIN {X 0,Y 291.02,Z 418.918,A -85,B 0,C 180,E1 -17439.126,E2 -17439.126} C_VEL
LIN {X 0,Y 288.803,Z 426.181,A -85,B 0,C 180,E1 -17440.445,E2 -17440.445} C_VEL
LIN {X 0,Y 286.829,Z 432.221,A -85,B 0,C 180,E1 -17441.789,E2 -17441.789} C_VEL
LIN {X 0,Y 284.587,Z 438.42,A -85,B 0,C 180,E1 -17443.495,E2 -17443.495} C_VEL
LIN {X 0,Y 282.162,Z 444.317,A -85,B 0,C 180,E1 -17445.571,E2 -17445.571} C_VEL
LIN {X 0,Y 280.062,Z 448.627,A -85,B 0,C 180,E1 -17447.677,E2 -17447.677} C_VEL
LIN {X 0,Y 278.573,Z 451.567,A -85,B 0,C 180,E1 -17449.821,E2 -17449.821} C_VEL
LIN {X 0,Y 277.583,Z 452.904,A -85,B 0,C 180,E1 -17451.255,E2 -17451.255} C_VEL
LIN {X 0,Y 276.793,Z 453.726,A -85,B 0,C 180,E1 -17452.699,E2 -17452.699} C_VEL
LIN {X 0,Y 276.321,Z 453.94,A -85,B 0,C 180,E1 -17454.154,E2 -17454.154} C_VEL
LIN {X 0,Y 275.938,Z 453.623,A -85,B 0,C 180,E1 -17455.611,E2 -17455.611} C_VEL
LIN {X 0,Y 275.609,Z 452.82,A -85,B 0,C 180,E1 -17457.069,E2 -17457.069} C_VEL
LIN {X 0,Y 275.394,Z 451.514,A -85,B 0,C 180,E1 -17458.53,E2 -17458.53} C_VEL
LIN {X 0,Y 275.294,Z 448.422,A -85,B 0,C 180,E1 -17460.724,E2 -17460.724} C_VEL
LIN {X 0,Y 275.452,Z 444.018,A -85,B 0,C 180,E1 -17462.917,E2 -17462.917} C_VEL
LIN {X 0,Y 275.565,Z 438.732,A -85,B 0,C 180,E1 -17464.891,E2 -17464.891} C_VEL
LIN {X 0,Y 275.865,Z 431.523,A -85,B 0,C 180,E1 -17466.942,E2 -17466.942} C_VEL
LIN {X 0,Y 276.227,Z 425.182,A -85,B 0,C 180,E1 -17468.404,E2 -17468.404} C_VEL
LIN {X 0,Y 276.632,Z 417.526,A -85,B 0,C 180,E1 -17469.866,E2 -17469.866} C_VEL
LIN {X 0,Y 277.014,Z 409.411,A -85,B 0,C 180,E1 -17471.146,E2 -17471.146} C_VEL
LIN {X 0,Y 277.62,Z 397.716,A -85,B 0,C 180,E1 -17472.604,E2 -17472.604} C_VEL
LIN {X 0,Y 278.08,Z 388.205,A -85,B 0,C 180,E1 -17473.511,E2 -17473.511} C_VEL
LIN {X 0,Y 278.451,Z 378.378,A -85,B 0,C 180,E1 -17474.238,E2 -17474.238} C_VEL
LIN {X 0,Y 278.752,Z 366.244,A -85,B 0,C 180,E1 -17474.875,E2 -17474.875} C_VEL
LIN {X 0,Y 279.866,Z 315.997,A -85,B 0,C 180,E1 -17476.895,E2 -17476.895} C_VEL
LIN {X 0,Y 277.437,Z 294.037,A -85,B 0,C 180,E1 -17477.831,E2 -17477.831} C_VEL
LIN {X 0,Y 277.528,Z 290.726,A -85,B 0,C 180,E1 -17479.116,E2 -17479.116} C_VEL
LIN {X 0,Y 277.231,Z 290.765,A -85,B 0,C 180,E1 -17484.125,E2 -17484.125} C_VEL
LIN {X 0,Y 277.221,Z 290.763,A -85,B 0,C 180,E1 -17487.46,E2 -17487.46} C_VEL
LIN {X 0,Y 277.213,Z 290.766,A -85,B 0,C 180,E1 -17490.457,E2 -17490.457} C_VEL
LIN {X 0,Y 277.228,Z 290.762,A -85,B 0,C 180,E1 -17493.887,E2 -17493.887} C_VEL
LIN {X 0,Y 277.212,Z 290.764,A -85,B 0,C 180,E1 -17497.466,E2 -17497.466} C_VEL
LIN {X 0,Y 277.152,Z 290.771,A -85,B 0,C 180,E1 -17501.234,E2 -17501.234} C_VEL
LIN {X 0,Y 277.17,Z 290.77,A -85,B 0,C 180,E1 -17505.219,E2 -17505.219} C_VEL
LIN {X 0,Y 277.188,Z 290.766,A -85,B 0,C 180,E1 -17509.505,E2 -17509.505} C_VEL
LIN {X 0,Y 277.231,Z 290.763,A -85,B 0,C 180,E1 -17512.522,E2 -17512.522} C_VEL
LIN {X 0,Y 277.211,Z 290.764,A -85,B 0,C 180,E1 -17516.097,E2 -17516.097} C_VEL
LIN {X 0,Y 277.225,Z 290.764,A -85,B 0,C 180,E1 -17519.532,E2 -17519.532} C_VEL
LIN {X 0,Y 277.312,Z 290.753,A -85,B 0,C 180,E1 -17522.857,E2 -17522.857} C_VEL
LIN {X 0,Y 277.254,Z 290.758,A -85,B 0,C 180,E1 -17526.07,E2 -17526.07} C_VEL
LIN {X 0,Y 277.298,Z 290.753,A -85,B 0,C 180,E1 -17530.76,E2 -17530.76} C_VEL
LIN {X 0,Y 277.369,Z 290.746,A -85,B 0,C 180,E1 -17535.32,E2 -17535.32} C_VEL
LIN {X 0,Y 277.458,Z 290.738,A -85,B 0,C 180,E1 -17539.785,E2 -17539.785} C_VEL
LIN {X 0,Y 277.598,Z 290.715,A -85,B 0,C 180,E1 -17542.725,E2 -17542.725} C_VEL
LIN {X 0,Y 277.776,Z 290.694,A -85,B 0,C 180,E1 -17548.548,E2 -17548.548} C_VEL
LIN {X 0,Y 277.775,Z 290.694,A -85,B 0,C 180,E1 -17551.447,E2 -17551.447} C_VEL
LIN {X 0,Y 277.594,Z 290.716,A -85,B 0,C 180,E1 -17557.27,E2 -17557.27} C_VEL
LIN {X 0,Y 277.454,Z 290.738,A -85,B 0,C 180,E1 -17560.211,E2 -17560.211} C_VEL
LIN {X 0,Y 277.363,Z 290.747,A -85,B 0,C 180,E1 -17564.675,E2 -17564.675} C_VEL
LIN {X 0,Y 277.29,Z 290.754,A -85,B 0,C 180,E1 -17569.235,E2 -17569.235} C_VEL
LIN {X 0,Y 277.24,Z 290.761,A -85,B 0,C 180,E1 -17574.159,E2 -17574.159} C_VEL
LIN {X 0,Y 277.273,Z 290.756,A -85,B 0,C 180,E1 -17577.506,E2 -17577.506} C_VEL
LIN {X 0,Y 277.223,Z 290.764,A -85,B 0,C 180,E1 -17580.484,E2 -17580.484} C_VEL
LIN {X 0,Y 277.205,Z 290.764,A -85,B 0,C 180,E1 -17583.898,E2 -17583.898} C_VEL
LIN {X 0,Y 277.238,Z 290.762,A -85,B 0,C 180,E1 -17587.47,E2 -17587.47} C_VEL
LIN {X 0,Y 277.248,Z 290.763,A -85,B 0,C 180,E1 -17591.226,E2 -17591.226} C_VEL
LIN {X 0,Y 277.244,Z 290.765,A -85,B 0,C 180,E1 -17595.213,E2 -17595.213} C_VEL
LIN {X 0,Y 277.254,Z 290.762,A -85,B 0,C 180,E1 -17599.5,E2 -17599.5} C_VEL
LIN {X 0,Y 277.246,Z 290.759,A -85,B 0,C 180,E1 -17602.539,E2 -17602.539} C_VEL
LIN {X 0,Y 277.217,Z 290.764,A -85,B 0,C 180,E1 -17606.111,E2 -17606.111} C_VEL
LIN {X 0,Y 277.227,Z 290.764,A -85,B 0,C 180,E1 -17609.545,E2 -17609.545} C_VEL
LIN {X 0,Y 277.324,Z 290.75,A -85,B 0,C 180,E1 -17612.87,E2 -17612.87} C_VEL
LIN {X 0,Y 277.266,Z 290.759,A -85,B 0,C 180,E1 -17616.083,E2 -17616.083} C_VEL
LIN {X 0,Y 277.283,Z 290.755,A -85,B 0,C 180,E1 -17620.771,E2 -17620.771} C_VEL
LIN {X 0,Y 277.384,Z 290.742,A -85,B 0,C 180,E1 -17625.332,E2 -17625.332} C_VEL
LIN {X 0,Y 277.435,Z 290.738,A -85,B 0,C 180,E1 -17629.794,E2 -17629.794} C_VEL
LIN {X 0,Y 277.596,Z 290.717,A -85,B 0,C 180,E1 -17632.735,E2 -17632.735} C_VEL
LIN {X 0,Y 277.797,Z 290.695,A -85,B 0,C 180,E1 -17638.558,E2 -17638.558} C_VEL
LIN {X 0,Y 277.794,Z 290.691,A -85,B 0,C 180,E1 -17641.457,E2 -17641.457} C_VEL
LIN {X 0,Y 277.588,Z 290.718,A -85,B 0,C 180,E1 -17647.295,E2 -17647.295} C_VEL
LIN {X 0,Y 277.444,Z 290.736,A -85,B 0,C 180,E1 -17650.22,E2 -17650.22} C_VEL
LIN {X 0,Y 277.356,Z 290.745,A -85,B 0,C 180,E1 -17653.597,E2 -17653.597} C_VEL
LIN {X 0,Y 276.651,Z 290.836,A -85,B 0,C 180,E1 -17654.808,E2 -17654.808} C_VEL
LIN {X 0,Y 273.752,Z 291.198,A -85,B 0,C 180,E1 -17656.779,E2 -17656.779} C_VEL
LIN {X 0,Y 271.319,Z 291.5,A -85,B 0,C 180,E1 -17658.381,E2 -17658.381} C_VEL
LIN {X 0,Y 270.292,Z 291.627,A -85,B 0,C 180,E1 -17659.624,E2 -17659.624} C_VEL
LIN {X 0,Y 270.217,Z 291.635,A -85,B 0,C 180,E1 -17660.045,E2 -17660.045} C_VEL
LIN {X 0,Y 270.175,Z 291.641,A -85,B 0,C 180,E1 -17664.602,E2 -17664.602} C_VEL
LIN {X 0,Y 270.195,Z 291.638,A -85,B 0,C 180,E1 -17667.924,E2 -17667.924} C_VEL
LIN {X 0,Y 270.174,Z 291.644,A -85,B 0,C 180,E1 -17671.356,E2 -17671.356} C_VEL
LIN {X 0,Y 270.198,Z 291.638,A -85,B 0,C 180,E1 -17674.913,E2 -17674.913} C_VEL
LIN {X 0,Y 270.202,Z 291.636,A -85,B 0,C 180,E1 -17678.717,E2 -17678.717} C_VEL
LIN {X 0,Y 270.152,Z 291.644,A -85,B 0,C 180,E1 -17683.25,E2 -17683.25} C_VEL
LIN {X 0,Y 270.156,Z 291.644,A -85,B 0,C 180,E1 -17687.443,E2 -17687.443} C_VEL
LIN {X 0,Y 270.185,Z 291.639,A -85,B 0,C 180,E1 -17691.374,E2 -17691.374} C_VEL
LIN {X 0,Y 270.206,Z 291.636,A -85,B 0,C 180,E1 -17695.099,E2 -17695.099} C_VEL
LIN {X 0,Y 270.182,Z 291.638,A -85,B 0,C 180,E1 -17699.146,E2 -17699.146} C_VEL
LIN {X 0,Y 270.415,Z 291.697,A -85,B 0,C 180,E1 -17703.731,E2 -17703.731} C_VEL
LIN {X 0,Y 271.635,Z 298.764,A -85,B 0,C 180,E1 -17706.36,E2 -17706.36} C_VEL
LIN {X 0,Y 270.852,Z 306.344,A -85,B 0,C 180,E1 -17709.099,E2 -17709.099} C_VEL
LIN {X 0,Y 270.029,Z 314.235,A -85,B 0,C 180,E1 -17711.951,E2 -17711.951} C_VEL
LIN {X 0,Y 270.787,Z 331.184,A -85,B 0,C 180,E1 -17712.711,E2 -17712.711} C_VEL
LIN {X 0,Y 272.468,Z 350.979,A -85,B 0,C 180,E1 -17713.568,E2 -17713.568} C_VEL
LIN {X 0,Y 271.453,Z 393.616,A -85,B 0,C 180,E1 -17715.429,E2 -17715.429} C_VEL
LIN {X 0,Y 271.014,Z 406.481,A -85,B 0,C 180,E1 -17716.315,E2 -17716.315} C_VEL
LIN {X 0,Y 270.517,Z 416.24,A -85,B 0,C 180,E1 -17717.245,E2 -17717.245} C_VEL
LIN {X 0,Y 269.898,Z 426.96,A -85,B 0,C 180,E1 -17718.551,E2 -17718.551} C_VEL
LIN {X 0,Y 269.497,Z 436.466,A -85,B 0,C 180,E1 -17720.054,E2 -17720.054} C_VEL
LIN {X 0,Y 269.196,Z 443.282,A -85,B 0,C 180,E1 -17721.369,E2 -17721.369} C_VEL
LIN {X 0,Y 268.996,Z 449.696,A -85,B 0,C 180,E1 -17722.851,E2 -17722.851} C_VEL
LIN {X 0,Y 268.832,Z 455.168,A -85,B 0,C 180,E1 -17724.377,E2 -17724.377} C_VEL
LIN {X 0,Y 268.737,Z 458.638,A -85,B 0,C 180,E1 -17725.503,E2 -17725.503} C_VEL
LIN {X 0,Y 268.61,Z 462.479,A -85,B 0,C 180,E1 -17727.003,E2 -17727.003} C_VEL
LIN {X 0,Y 268.655,Z 466.791,A -85,B 0,C 180,E1 -17729.253,E2 -17729.253} C_VEL
LIN {X 0,Y 268.708,Z 467.949,A -85,B 0,C 180,E1 -17730.003,E2 -17730.003} C_VEL
LIN {X 0,Y 268.288,Z 469.681,A -85,B 0,C 180,E1 -17731.504,E2 -17731.504} C_VEL
LIN {X 0,Y 268.281,Z 470.936,A -85,B 0,C 180,E1 -17733.006,E2 -17733.006} C_VEL
LIN {X 0,Y 268.296,Z 471.691,A -85,B 0,C 180,E1 -17734.51,E2 -17734.51} C_VEL
LIN {X 0,Y 268.37,Z 471.872,A -85,B 0,C 180,E1 -17736.015,E2 -17736.015} C_VEL
LIN {X 0,Y 268.671,Z 471.48,A -85,B 0,C 180,E1 -17737.518,E2 -17737.518} C_VEL
LIN {X 0,Y 269.123,Z 470.629,A -85,B 0,C 180,E1 -17739.017,E2 -17739.017} C_VEL
LIN {X 0,Y 269.829,Z 469.304,A -85,B 0,C 180,E1 -17740.508,E2 -17740.508} C_VEL
LIN {X 0,Y 271.266,Z 466.215,A -85,B 0,C 180,E1 -17742.724,E2 -17742.724} C_VEL
LIN {X 0,Y 273.261,Z 461.887,A -85,B 0,C 180,E1 -17744.906,E2 -17744.906} C_VEL
LIN {X 0,Y 275.514,Z 456.211,A -85,B 0,C 180,E1 -17747.061,E2 -17747.061} C_VEL
LIN {X 0,Y 278.362,Z 448.68,A -85,B 0,C 180,E1 -17749.163,E2 -17749.163} C_VEL
LIN {X 0,Y 281.185,Z 440.874,A -85,B 0,C 180,E1 -17750.867,E2 -17750.867} C_VEL
LIN {X 0,Y 284.379,Z 431.255,A -85,B 0,C 180,E1 -17752.526,E2 -17752.526} C_VEL
LIN {X 0,Y 287.188,Z 421.427,A -85,B 0,C 180,E1 -17753.817,E2 -17753.817} C_VEL
LIN {X 0,Y 289.948,Z 410.682,A -85,B 0,C 180,E1 -17754.909,E2 -17754.909} C_VEL
LIN {X 0,Y 292.496,Z 398.838,A -85,B 0,C 180,E1 -17755.819,E2 -17755.819} C_VEL
LIN {X 0,Y 294.29,Z 387.535,A -85,B 0,C 180,E1 -17756.46,E2 -17756.46} C_VEL
LIN {X 0,Y 297.487,Z 360.079,A -85,B 0,C 180,E1 -17757.701,E2 -17757.701} C_VEL
LIN {X 0,Y 296.729,Z 349.897,A -85,B 0,C 180,E1 -17758.666,E2 -17758.666} C_VEL
LIN {X 0,Y 295.289,Z 338.793,A -85,B 0,C 180,E1 -17759.956,E2 -17759.956} C_VEL
LIN {X 0,Y 292.217,Z 331.635,A -85,B 0,C 180,E1 -17761.57,E2 -17761.57} C_VEL
LIN {X 0,Y 290.772,Z 328.614,A -85,B 0,C 180,E1 -17762.358,E2 -17762.358} C_VEL
LIN {X 0,Y 288.284,Z 323.542,A -85,B 0,C 180,E1 -17763.896,E2 -17763.896} C_VEL
LIN {X 0,Y 284.716,Z 317.195,A -85,B 0,C 180,E1 -17766.446,E2 -17766.446} C_VEL
LIN {X 0,Y 281.613,Z 312.008,A -85,B 0,C 180,E1 -17769.609,E2 -17769.609} C_VEL
LIN {X 0,Y 280.281,Z 309.485,A -85,B 0,C 180,E1 -17771.846,E2 -17771.846} C_VEL
LIN {X 0,Y 279.522,Z 308.111,A -85,B 0,C 180,E1 -17774.402,E2 -17774.402} C_VEL
LIN {X 0,Y 279.839,Z 307.869,A -85,B 0,C 180,E1 -17777.573,E2 -17777.573} C_VEL
LIN {X 0,Y 281.784,Z 309.845,A -85,B 0,C 180,E1 -17780.94,E2 -17780.94} C_VEL
LIN {X 0,Y 283.656,Z 311.625,A -85,B 0,C 180,E1 -17782.84,E2 -17782.84} C_VEL
LIN {X 0,Y 286.826,Z 315.815,A -85,B 0,C 180,E1 -17785.362,E2 -17785.362} C_VEL
LIN {X 0,Y 290.833,Z 321.721,A -85,B 0,C 180,E1 -17787.837,E2 -17787.837} C_VEL
LIN {X 0,Y 293.739,Z 326.462,A -85,B 0,C 180,E1 -17789.347,E2 -17789.347} C_VEL
LIN {X 0,Y 297.365,Z 332.932,A -85,B 0,C 180,E1 -17791.037,E2 -17791.037} C_VEL
LIN {X 0,Y 299.745,Z 338.167,A -85,B 0,C 180,E1 -17792.109,E2 -17792.109} C_VEL
LIN {X 0,Y 294.71,Z 378.239,A -85,B 0,C 180,E1 -17793.91,E2 -17793.91} C_VEL
LIN {X 0,Y 292.635,Z 390.69,A -85,B 0,C 180,E1 -17794.762,E2 -17794.762} C_VEL
LIN {X 0,Y 290.834,Z 399.324,A -85,B 0,C 180,E1 -17795.548,E2 -17795.548} C_VEL
LIN {X 0,Y 288.166,Z 410.457,A -85,B 0,C 180,E1 -17796.836,E2 -17796.836} C_VEL
LIN {X 0,Y 285.363,Z 420.138,A -85,B 0,C 180,E1 -17798.314,E2 -17798.314} C_VEL
LIN {X 0,Y 282.974,Z 427.209,A -85,B 0,C 180,E1 -17799.646,E2 -17799.646} C_VEL
LIN {X 0,Y 280.847,Z 433.077,A -85,B 0,C 180,E1 -17801.009,E2 -17801.009} C_VEL
LIN {X 0,Y 278.445,Z 439.194,A -85,B 0,C 180,E1 -17802.742,E2 -17802.742} C_VEL
LIN {X 0,Y 276.252,Z 444.116,A -85,B 0,C 180,E1 -17804.5,E2 -17804.5} C_VEL
LIN {X 0,Y 273.916,Z 448.599,A -85,B 0,C 180,E1 -17806.642,E2 -17806.642} C_VEL
LIN {X 0,Y 272.626,Z 450.809,A -85,B 0,C 180,E1 -17808.092,E2 -17808.092} C_VEL
LIN {X 0,Y 271.658,Z 452.415,A -85,B 0,C 180,E1 -17809.559,E2 -17809.559} C_VEL
LIN {X 0,Y 270.596,Z 453.538,A -85,B 0,C 180,E1 -17811.028,E2 -17811.028} C_VEL
LIN {X 0,Y 269.78,Z 454.16,A -85,B 0,C 180,E1 -17812.509,E2 -17812.509} C_VEL
LIN {X 0,Y 269.269,Z 454.285,A -85,B 0,C 180,E1 -17814,E2 -17814} C_VEL
LIN {X 0,Y 268.886,Z 453.815,A -85,B 0,C 180,E1 -17815.495,E2 -17815.495} C_VEL
LIN {X 0,Y 268.544,Z 452.81,A -85,B 0,C 180,E1 -17816.992,E2 -17816.992} C_VEL
LIN {X 0,Y 268.257,Z 450.379,A -85,B 0,C 180,E1 -17819.242,E2 -17819.242} C_VEL
LIN {X 0,Y 268.246,Z 446.641,A -85,B 0,C 180,E1 -17821.494,E2 -17821.494} C_VEL
LIN {X 0,Y 268.487,Z 441.372,A -85,B 0,C 180,E1 -17823.744,E2 -17823.744} C_VEL
LIN {X 0,Y 268.534,Z 435.976,A -85,B 0,C 180,E1 -17825.544,E2 -17825.544} C_VEL
LIN {X 0,Y 268.933,Z 428.704,A -85,B 0,C 180,E1 -17827.5,E2 -17827.5} C_VEL
LIN {X 0,Y 269.373,Z 419.715,A -85,B 0,C 180,E1 -17829.377,E2 -17829.377} C_VEL
LIN {X 0,Y 269.809,Z 410.707,A -85,B 0,C 180,E1 -17830.877,E2 -17830.877} C_VEL
LIN {X 0,Y 270.377,Z 401.035,A -85,B 0,C 180,E1 -17832.184,E2 -17832.184} C_VEL
LIN {X 0,Y 270.905,Z 389.19,A -85,B 0,C 180,E1 -17833.398,E2 -17833.398} C_VEL
LIN {X 0,Y 271.302,Z 379.592,A -85,B 0,C 180,E1 -17834.142,E2 -17834.142} C_VEL
LIN {X 0,Y 271.623,Z 368.019,A -85,B 0,C 180,E1 -17834.795,E2 -17834.795} C_VEL
LIN {X 0,Y 272.813,Z 316.66,A -85,B 0,C 180,E1 -17836.966,E2 -17836.966} C_VEL
LIN {X 0,Y 270.41,Z 294.851,A -85,B 0,C 180,E1 -17837.92,E2 -17837.92} C_VEL
LIN {X 0,Y 270.374,Z 294.001,A -85,B 0,C 180,E1 -17838.004,E2 -17838.004} C_VEL
LIN {X 0,Y 270.408,Z 291.613,A -85,B 0,C 180,E1 -17838.949,E2 -17838.949} C_VEL
LIN {X 0,Y 270.183,Z 291.638,A -85,B 0,C 180,E1 -17842.956,E2 -17842.956} C_VEL
LIN {X 0,Y 270.166,Z 291.647,A -85,B 0,C 180,E1 -17846.236,E2 -17846.236} C_VEL
LIN {X 0,Y 270.141,Z 291.644,A -85,B 0,C 180,E1 -17849.613,E2 -17849.613} C_VEL
LIN {X 0,Y 270.197,Z 291.637,A -85,B 0,C 180,E1 -17853.657,E2 -17853.657} C_VEL
LIN {X 0,Y 270.178,Z 291.643,A -85,B 0,C 180,E1 -17856.735,E2 -17856.735} C_VEL
LIN {X 0,Y 270.11,Z 291.649,A -85,B 0,C 180,E1 -17861.011,E2 -17861.011} C_VEL
LIN {X 0,Y 270.119,Z 291.651,A -85,B 0,C 180,E1 -17864.613,E2 -17864.613} C_VEL
LIN {X 0,Y 270.134,Z 291.645,A -85,B 0,C 180,E1 -17867.432,E2 -17867.432} C_VEL
LIN {X 0,Y 270.176,Z 291.641,A -85,B 0,C 180,E1 -17871.366,E2 -17871.366} C_VEL
LIN {X 0,Y 270.166,Z 291.646,A -85,B 0,C 180,E1 -17875.087,E2 -17875.087} C_VEL
LIN {X 0,Y 270.147,Z 291.647,A -85,B 0,C 180,E1 -17879.13,E2 -17879.13} C_VEL
LIN {X 0,Y 270.223,Z 291.634,A -85,B 0,C 180,E1 -17882.14,E2 -17882.14} C_VEL
LIN {X 0,Y 270.195,Z 291.64,A -85,B 0,C 180,E1 -17885.532,E2 -17885.532} C_VEL
LIN {X 0,Y 270.256,Z 291.63,A -85,B 0,C 180,E1 -17890.239,E2 -17890.239} C_VEL
LIN {X 0,Y 270.337,Z 291.62,A -85,B 0,C 180,E1 -17894.929,E2 -17894.929} C_VEL
LIN {X 0,Y 270.394,Z 291.616,A -85,B 0,C 180,E1 -17899.515,E2 -17899.515} C_VEL
LIN {X 0,Y 270.556,Z 291.593,A -85,B 0,C 180,E1 -17902.535,E2 -17902.535} C_VEL
LIN {X 0,Y 270.742,Z 291.571,A -85,B 0,C 180,E1 -17908.51,E2 -17908.51} C_VEL
LIN {X 0,Y 270.741,Z 291.571,A -85,B 0,C 180,E1 -17911.485,E2 -17911.485} C_VEL
LIN {X 0,Y 270.552,Z 291.593,A -85,B 0,C 180,E1 -17917.46,E2 -17917.46} C_VEL
LIN {X 0,Y 270.39,Z 291.617,A -85,B 0,C 180,E1 -17920.48,E2 -17920.48} C_VEL
LIN {X 0,Y 270.331,Z 291.621,A -85,B 0,C 180,E1 -17925.066,E2 -17925.066} C_VEL
LIN {X 0,Y 270.248,Z 291.631,A -85,B 0,C 180,E1 -17929.757,E2 -17929.757} C_VEL
LIN {X 0,Y 270.187,Z 291.642,A -85,B 0,C 180,E1 -17934.591,E2 -17934.591} C_VEL
LIN {X 0,Y 270.222,Z 291.635,A -85,B 0,C 180,E1 -17937.911,E2 -17937.911} C_VEL
LIN {X 0,Y 270.135,Z 291.645,A -85,B 0,C 180,E1 -17941.351,E2 -17941.351} C_VEL
LIN {X 0,Y 270.167,Z 291.646,A -85,B 0,C 180,E1 -17944.907,E2 -17944.907} C_VEL
LIN {X 0,Y 270.177,Z 291.642,A -85,B 0,C 180,E1 -17948.721,E2 -17948.721} C_VEL
LIN {X 0,Y 270.211,Z 291.636,A -85,B 0,C 180,E1 -17952.546,E2 -17952.546} C_VEL
LIN {X 0,Y 270.189,Z 291.639,A -85,B 0,C 180,E1 -17956.741,E2 -17956.741} C_VEL
LIN {X 0,Y 270.208,Z 291.639,A -85,B 0,C 180,E1 -17959.453,E2 -17959.453} C_VEL
LIN {X 0,Y 270.217,Z 291.638,A -85,B 0,C 180,E1 -17963.728,E2 -17963.728} C_VEL
LIN {X 0,Y 270.167,Z 291.641,A -85,B 0,C 180,E1 -17966.899,E2 -17966.899} C_VEL
LIN {X 0,Y 270.161,Z 291.642,A -85,B 0,C 180,E1 -17970.389,E2 -17970.389} C_VEL
LIN {X 0,Y 270.228,Z 291.639,A -85,B 0,C 180,E1 -17973.77,E2 -17973.77} C_VEL
LIN {X 0,Y 270.177,Z 291.639,A -85,B 0,C 180,E1 -17977.043,E2 -17977.043} C_VEL
LIN {X 0,Y 270.226,Z 291.637,A -85,B 0,C 180,E1 -17980.248,E2 -17980.248} C_VEL
LIN {X 0,Y 270.352,Z 291.617,A -85,B 0,C 180,E1 -17984.941,E2 -17984.941} C_VEL
LIN {X 0,Y 270.387,Z 291.614,A -85,B 0,C 180,E1 -17989.525,E2 -17989.525} C_VEL
LIN {X 0,Y 270.555,Z 291.596,A -85,B 0,C 180,E1 -17992.545,E2 -17992.545} C_VEL
LIN {X 0,Y 270.761,Z 291.572,A -85,B 0,C 180,E1 -17998.52,E2 -17998.52} C_VEL
LIN {X 0,Y 270.759,Z 291.567,A -85,B 0,C 180,E1 -18001.495,E2 -18001.495} C_VEL
LIN {X 0,Y 270.551,Z 291.594,A -85,B 0,C 180,E1 -18007.47,E2 -18007.47} C_VEL
LIN {X 0,Y 270.396,Z 291.615,A -85,B 0,C 180,E1 -18010.49,E2 -18010.49} C_VEL
LIN {X 0,Y 270.331,Z 291.624,A -85,B 0,C 180,E1 -18015.076,E2 -18015.076} C_VEL
LIN {X 0,Y 270.217,Z 291.635,A -85,B 0,C 180,E1 -18020.045,E2 -18020.045} C_VEL
LIN {X 0,Y 269.554,Z 291.72,A -85,B 0,C 180,E1 -18021.289,E2 -18021.289} C_VEL
LIN {X 0,Y 266.651,Z 292.082,A -85,B 0,C 180,E1 -18023.314,E2 -18023.314} C_VEL
LIN {X 0,Y 264.197,Z 292.387,A -85,B 0,C 180,E1 -18024.961,E2 -18024.961} C_VEL
LIN {X 0,Y 263.173,Z 292.513,A -85,B 0,C 180,E1 -18026.239,E2 -18026.239} C_VEL
LIN {X 0,Y 263.106,Z 292.522,A -85,B 0,C 180,E1 -18026.672,E2 -18026.672} C_VEL
LIN {X 0,Y 263.124,Z 292.518,A -85,B 0,C 180,E1 -18030.504,E2 -18030.504} C_VEL
LIN {X 0,Y 263.154,Z 292.515,A -85,B 0,C 180,E1 -18034.121,E2 -18034.121} C_VEL
LIN {X 0,Y 263.123,Z 292.52,A -85,B 0,C 180,E1 -18037.91,E2 -18037.91} C_VEL
LIN {X 0,Y 263.084,Z 292.526,A -85,B 0,C 180,E1 -18041.909,E2 -18041.909} C_VEL
LIN {X 0,Y 263.085,Z 292.525,A -85,B 0,C 180,E1 -18046.167,E2 -18046.167} C_VEL
LIN {X 0,Y 263.121,Z 292.518,A -85,B 0,C 180,E1 -18050.776,E2 -18050.776} C_VEL
LIN {X 0,Y 263.164,Z 292.519,A -85,B 0,C 180,E1 -18054.022,E2 -18054.022} C_VEL
LIN {X 0,Y 263.136,Z 292.518,A -85,B 0,C 180,E1 -18057.716,E2 -18057.716} C_VEL
LIN {X 0,Y 263.362,Z 292.489,A -85,B 0,C 180,E1 -18063.453,E2 -18063.453} C_VEL
LIN {X 0,Y 263.387,Z 292.507,A -85,B 0,C 180,E1 -18063.776,E2 -18063.776} C_VEL
LIN {X 0,Y 264.53,Z 298.642,A -85,B 0,C 180,E1 -18066.125,E2 -18066.125} C_VEL
LIN {X 0,Y 263.859,Z 305.81,A -85,B 0,C 180,E1 -18068.799,E2 -18068.799} C_VEL
LIN {X 0,Y 262.966,Z 314.03,A -85,B 0,C 180,E1 -18071.852,E2 -18071.852} C_VEL
LIN {X 0,Y 263.673,Z 331.257,A -85,B 0,C 180,E1 -18072.654,E2 -18072.654} C_VEL
LIN {X 0,Y 265.376,Z 350.706,A -85,B 0,C 180,E1 -18073.528,E2 -18073.528} C_VEL
LIN {X 0,Y 264.36,Z 393.607,A -85,B 0,C 180,E1 -18075.472,E2 -18075.472} C_VEL
LIN {X 0,Y 263.962,Z 405.815,A -85,B 0,C 180,E1 -18076.335,E2 -18076.335} C_VEL
LIN {X 0,Y 263.443,Z 415.616,A -85,B 0,C 180,E1 -18077.289,E2 -18077.289} C_VEL
LIN {X 0,Y 262.917,Z 424.96,A -85,B 0,C 180,E1 -18078.438,E2 -18078.438} C_VEL
LIN {X 0,Y 262.504,Z 434.96,A -85,B 0,C 180,E1 -18079.981,E2 -18079.981} C_VEL
LIN {X 0,Y 262.137,Z 442.811,A -85,B 0,C 180,E1 -18081.523,E2 -18081.523} C_VEL
LIN {X 0,Y 261.97,Z 449.305,A -85,B 0,C 180,E1 -18083.07,E2 -18083.07} C_VEL
LIN {X 0,Y 261.816,Z 454.712,A -85,B 0,C 180,E1 -18084.624,E2 -18084.624} C_VEL
LIN {X 0,Y 261.666,Z 459.116,A -85,B 0,C 180,E1 -18086.153,E2 -18086.153} C_VEL
LIN {X 0,Y 261.615,Z 464.325,A -85,B 0,C 180,E1 -18088.463,E2 -18088.463} C_VEL
LIN {X 0,Y 261.684,Z 466.931,A -85,B 0,C 180,E1 -18090.003,E2 -18090.003} C_VEL
LIN {X 0,Y 261.248,Z 468.877,A -85,B 0,C 180,E1 -18091.544,E2 -18091.544} C_VEL
LIN {X 0,Y 261.216,Z 470.333,A -85,B 0,C 180,E1 -18093.087,E2 -18093.087} C_VEL
LIN {X 0,Y 261.212,Z 471.37,A -85,B 0,C 180,E1 -18095.391,E2 -18095.391} C_VEL
LIN {X 0,Y 261.616,Z 471.29,A -85,B 0,C 180,E1 -18097.722,E2 -18097.722} C_VEL
LIN {X 0,Y 262.115,Z 470.656,A -85,B 0,C 180,E1 -18099.26,E2 -18099.26} C_VEL
LIN {X 0,Y 262.844,Z 469.482,A -85,B 0,C 180,E1 -18100.79,E2 -18100.79} C_VEL
LIN {X 0,Y 264.362,Z 466.736,A -85,B 0,C 180,E1 -18103.062,E2 -18103.062} C_VEL
LIN {X 0,Y 266.462,Z 462.679,A -85,B 0,C 180,E1 -18105.295,E2 -18105.295} C_VEL
LIN {X 0,Y 268.375,Z 458.277,A -85,B 0,C 180,E1 -18107.136,E2 -18107.136} C_VEL
LIN {X 0,Y 270.752,Z 452.834,A -85,B 0,C 180,E1 -18108.936,E2 -18108.936} C_VEL
LIN {X 0,Y 273.569,Z 446.13,A -85,B 0,C 180,E1 -18110.688,E2 -18110.688} C_VEL
LIN {X 0,Y 276.719,Z 437.882,A -85,B 0,C 180,E1 -18112.396,E2 -18112.396} C_VEL
LIN {X 0,Y 279.809,Z 428.591,A -85,B 0,C 180,E1 -18113.894,E2 -18113.894} C_VEL
LIN {X 0,Y 282.555,Z 419.808,A -85,B 0,C 180,E1 -18115.016,E2 -18115.016} C_VEL
LIN {X 0,Y 285.492,Z 408.995,A -85,B 0,C 180,E1 -18116.108,E2 -18116.108} C_VEL
LIN {X 0,Y 287.977,Z 397.696,A -85,B 0,C 180,E1 -18116.939,E2 -18116.939} C_VEL
LIN {X 0,Y 289.967,Z 385.341,A -85,B 0,C 180,E1 -18117.633,E2 -18117.633} C_VEL
LIN {X 0,Y 292.963,Z 361.902,A -85,B 0,C 180,E1 -18118.709,E2 -18118.709} C_VEL
LIN {X 0,Y 292.299,Z 351.675,A -85,B 0,C 180,E1 -18119.727,E2 -18119.727} C_VEL
LIN {X 0,Y 291.317,Z 343.121,A -85,B 0,C 180,E1 -18120.79,E2 -18120.79} C_VEL
LIN {X 0,Y 288.877,Z 337.064,A -85,B 0,C 180,E1 -18122.178,E2 -18122.178} C_VEL
LIN {X 0,Y 287.394,Z 333.725,A -85,B 0,C 180,E1 -18123.112,E2 -18123.112} C_VEL
LIN {X 0,Y 285.278,Z 329.266,A -85,B 0,C 180,E1 -18124.517,E2 -18124.517} C_VEL
LIN {X 0,Y 282.344,Z 323.573,A -85,B 0,C 180,E1 -18126.856,E2 -18126.856} C_VEL
LIN {X 0,Y 279.587,Z 318.667,A -85,B 0,C 180,E1 -18129.87,E2 -18129.87} C_VEL
LIN {X 0,Y 278.4,Z 316.243,A -85,B 0,C 180,E1 -18132.038,E2 -18132.038} C_VEL
LIN {X 0,Y 277.742,Z 314.985,A -85,B 0,C 180,E1 -18134.433,E2 -18134.433} C_VEL
LIN {X 0,Y 278.093,Z 314.792,A -85,B 0,C 180,E1 -18137.667,E2 -18137.667} C_VEL
LIN {X 0,Y 279.933,Z 316.707,A -85,B 0,C 180,E1 -18140.885,E2 -18140.885} C_VEL
LIN {X 0,Y 281.563,Z 318.375,A -85,B 0,C 180,E1 -18142.628,E2 -18142.628} C_VEL
LIN {X 0,Y 284.967,Z 323.194,A -85,B 0,C 180,E1 -18145.436,E2 -18145.436} C_VEL
LIN {X 0,Y 288.204,Z 328.159,A -85,B 0,C 180,E1 -18147.503,E2 -18147.503} C_VEL
LIN {X 0,Y 291.261,Z 333.417,A -85,B 0,C 180,E1 -18149.185,E2 -18149.185} C_VEL
LIN {X 0,Y 294.481,Z 339.791,A -85,B 0,C 180,E1 -18150.796,E2 -18150.796} C_VEL
LIN {X 0,Y 295.141,Z 341.582,A -85,B 0,C 180,E1 -18151.131,E2 -18151.131} C_VEL
LIN {X 0,Y 290.06,Z 379.11,A -85,B 0,C 180,E1 -18152.876,E2 -18152.876} C_VEL
LIN {X 0,Y 287.853,Z 391.318,A -85,B 0,C 180,E1 -18153.729,E2 -18153.729} C_VEL
LIN {X 0,Y 285.588,Z 401.473,A -85,B 0,C 180,E1 -18154.68,E2 -18154.68} C_VEL
LIN {X 0,Y 282.745,Z 412.107,A -85,B 0,C 180,E1 -18155.976,E2 -18155.976} C_VEL
LIN {X 0,Y 280.394,Z 419.553,A -85,B 0,C 180,E1 -18157.132,E2 -18157.132} C_VEL
LIN {X 0,Y 277.238,Z 428.335,A -85,B 0,C 180,E1 -18158.817,E2 -18158.817} C_VEL
LIN {X 0,Y 274.45,Z 435.453,A -85,B 0,C 180,E1 -18160.549,E2 -18160.549} C_VEL
LIN {X 0,Y 271.412,Z 442.07,A -85,B 0,C 180,E1 -18162.669,E2 -18162.669} C_VEL
LIN {X 0,Y 268.721,Z 447.128,A -85,B 0,C 180,E1 -18164.832,E2 -18164.832} C_VEL
LIN {X 0,Y 267.108,Z 449.747,A -85,B 0,C 180,E1 -18166.295,E2 -18166.295} C_VEL
LIN {X 0,Y 265.757,Z 451.794,A -85,B 0,C 180,E1 -18167.779,E2 -18167.779} C_VEL
LIN {X 0,Y 264.75,Z 453.271,A -85,B 0,C 180,E1 -18169.284,E2 -18169.284} C_VEL
LIN {X 0,Y 263.621,Z 454.174,A -85,B 0,C 180,E1 -18170.788,E2 -18170.788} C_VEL
LIN {X 0,Y 262.772,Z 454.572,A -85,B 0,C 180,E1 -18172.308,E2 -18172.308} C_VEL
LIN {X 0,Y 262.223,Z 454.489,A -85,B 0,C 180,E1 -18173.838,E2 -18173.838} C_VEL
LIN {X 0,Y 261.814,Z 453.923,A -85,B 0,C 180,E1 -18175.373,E2 -18175.373} C_VEL
LIN {X 0,Y 261.481,Z 452.774,A -85,B 0,C 180,E1 -18176.911,E2 -18176.911} C_VEL
LIN {X 0,Y 261.182,Z 450.078,A -85,B 0,C 180,E1 -18179.221,E2 -18179.221} C_VEL
LIN {X 0,Y 261.176,Z 445.982,A -85,B 0,C 180,E1 -18181.534,E2 -18181.534} C_VEL
LIN {X 0,Y 261.43,Z 440.451,A -85,B 0,C 180,E1 -18183.846,E2 -18183.846} C_VEL
LIN {X 0,Y 261.575,Z 433.163,A -85,B 0,C 180,E1 -18186.161,E2 -18186.161} C_VEL
LIN {X 0,Y 262.018,Z 425.309,A -85,B 0,C 180,E1 -18188.087,E2 -18188.087} C_VEL
LIN {X 0,Y 262.421,Z 417.623,A -85,B 0,C 180,E1 -18189.627,E2 -18189.627} C_VEL
LIN {X 0,Y 262.901,Z 408.26,A -85,B 0,C 180,E1 -18191.167,E2 -18191.167} C_VEL
LIN {X 0,Y 263.416,Z 397.676,A -85,B 0,C 180,E1 -18192.511,E2 -18192.511} C_VEL
LIN {X 0,Y 263.868,Z 388.04,A -85,B 0,C 180,E1 -18193.468,E2 -18193.468} C_VEL
LIN {X 0,Y 264.319,Z 376.721,A -85,B 0,C 180,E1 -18194.327,E2 -18194.327} C_VEL
LIN {X 0,Y 264.702,Z 360.041,A -85,B 0,C 180,E1 -18195.142,E2 -18195.142} C_VEL
LIN {X 0,Y 265.662,Z 316.507,A -85,B 0,C 180,E1 -18197.045,E2 -18197.045} C_VEL
LIN {X 0,Y 263.349,Z 295.244,A -85,B 0,C 180,E1 -18198.013,E2 -18198.013} C_VEL
LIN {X 0,Y 263.312,Z 294.393,A -85,B 0,C 180,E1 -18198.066,E2 -18198.066} C_VEL
LIN {X 0,Y 263.354,Z 292.492,A -85,B 0,C 180,E1 -18198.87,E2 -18198.87} C_VEL
LIN {X 0,Y 263.148,Z 292.518,A -85,B 0,C 180,E1 -18201.947,E2 -18201.947} C_VEL
LIN {X 0,Y 263.11,Z 292.52,A -85,B 0,C 180,E1 -18205.291,E2 -18205.291} C_VEL
LIN {X 0,Y 263.104,Z 292.522,A -85,B 0,C 180,E1 -18208.728,E2 -18208.728} C_VEL
LIN {X 0,Y 263.109,Z 292.522,A -85,B 0,C 180,E1 -18212.28,E2 -18212.28} C_VEL
LIN {X 0,Y 263.134,Z 292.519,A -85,B 0,C 180,E1 -18215.975,E2 -18215.975} C_VEL
LIN {X 0,Y 263.049,Z 292.527,A -85,B 0,C 180,E1 -18219.87,E2 -18219.87} C_VEL
LIN {X 0,Y 263.056,Z 292.527,A -85,B 0,C 180,E1 -18223.984,E2 -18223.984} C_VEL
LIN {X 0,Y 263.09,Z 292.524,A -85,B 0,C 180,E1 -18228.4,E2 -18228.4} C_VEL
LIN {X 0,Y 263.127,Z 292.518,A -85,B 0,C 180,E1 -18232.095,E2 -18232.095} C_VEL
LIN {X 0,Y 263.117,Z 292.519,A -85,B 0,C 180,E1 -18235.878,E2 -18235.878} C_VEL
LIN {X 0,Y 263.092,Z 292.524,A -85,B 0,C 180,E1 -18239.497,E2 -18239.497} C_VEL
LIN {X 0,Y 263.149,Z 292.519,A -85,B 0,C 180,E1 -18242.995,E2 -18242.995} C_VEL
LIN {X 0,Y 263.112,Z 292.519,A -85,B 0,C 180,E1 -18246.378,E2 -18246.378} C_VEL
LIN {X 0,Y 263.219,Z 292.51,A -85,B 0,C 180,E1 -18249.687,E2 -18249.687} C_VEL
LIN {X 0,Y 263.284,Z 292.498,A -85,B 0,C 180,E1 -18254.516,E2 -18254.516} C_VEL
LIN {X 0,Y 263.326,Z 292.494,A -85,B 0,C 180,E1 -18259.23,E2 -18259.23} C_VEL
LIN {X 0,Y 263.519,Z 292.47,A -85,B 0,C 180,E1 -18262.334,E2 -18262.334} C_VEL
LIN {X 0,Y 263.707,Z 292.447,A -85,B 0,C 180,E1 -18268.47,E2 -18268.47} C_VEL
LIN {X 0,Y 263.707,Z 292.447,A -85,B 0,C 180,E1 -18271.525,E2 -18271.525} C_VEL
LIN {X 0,Y 263.515,Z 292.471,A -85,B 0,C 180,E1 -18277.661,E2 -18277.661} C_VEL
LIN {X 0,Y 263.322,Z 292.495,A -85,B 0,C 180,E1 -18280.765,E2 -18280.765} C_VEL
LIN {X 0,Y 263.278,Z 292.499,A -85,B 0,C 180,E1 -18285.479,E2 -18285.479} C_VEL
LIN {X 0,Y 263.211,Z 292.511,A -85,B 0,C 180,E1 -18290.308,E2 -18290.308} C_VEL
LIN {X 0,Y 263.142,Z 292.517,A -85,B 0,C 180,E1 -18295.295,E2 -18295.295} C_VEL
LIN {X 0,Y 263.13,Z 292.523,A -85,B 0,C 180,E1 -18298.732,E2 -18298.732} C_VEL
LIN {X 0,Y 263.085,Z 292.522,A -85,B 0,C 180,E1 -18302.291,E2 -18302.291} C_VEL
LIN {X 0,Y 263.141,Z 292.517,A -85,B 0,C 180,E1 -18305.982,E2 -18305.982} C_VEL
LIN {X 0,Y 263.116,Z 292.518,A -85,B 0,C 180,E1 -18309.866,E2 -18309.866} C_VEL
LIN {X 0,Y 263.148,Z 292.516,A -85,B 0,C 180,E1 -18313.869,E2 -18313.869} C_VEL
LIN {X 0,Y 263.171,Z 292.512,A -85,B 0,C 180,E1 -18318.39,E2 -18318.39} C_VEL
LIN {X 0,Y 263.165,Z 292.516,A -85,B 0,C 180,E1 -18323.237,E2 -18323.237} C_VEL
LIN {X 0,Y 263.147,Z 292.517,A -85,B 0,C 180,E1 -18325.896,E2 -18325.896} C_VEL
LIN {X 0,Y 263.106,Z 292.523,A -85,B 0,C 180,E1 -18329.512,E2 -18329.512} C_VEL
LIN {X 0,Y 263.158,Z 292.515,A -85,B 0,C 180,E1 -18333.009,E2 -18333.009} C_VEL
LIN {X 0,Y 263.122,Z 292.518,A -85,B 0,C 180,E1 -18336.391,E2 -18336.391} C_VEL
LIN {X 0,Y 263.208,Z 292.51,A -85,B 0,C 180,E1 -18339.698,E2 -18339.698} C_VEL
LIN {X 0,Y 263.298,Z 292.497,A -85,B 0,C 180,E1 -18344.528,E2 -18344.528} C_VEL
LIN {X 0,Y 263.327,Z 292.493,A -85,B 0,C 180,E1 -18349.241,E2 -18349.241} C_VEL
LIN {X 0,Y 263.516,Z 292.474,A -85,B 0,C 180,E1 -18352.345,E2 -18352.345} C_VEL
LIN {X 0,Y 263.724,Z 292.449,A -85,B 0,C 180,E1 -18358.481,E2 -18358.481} C_VEL
LIN {X 0,Y 263.723,Z 292.444,A -85,B 0,C 180,E1 -18361.535,E2 -18361.535} C_VEL
LIN {X 0,Y 263.515,Z 292.47,A -85,B 0,C 180,E1 -18367.671,E2 -18367.671} C_VEL
LIN {X 0,Y 263.334,Z 292.497,A -85,B 0,C 180,E1 -18370.774,E2 -18370.774} C_VEL
LIN {X 0,Y 263.281,Z 292.5,A -85,B 0,C 180,E1 -18375.489,E2 -18375.489} C_VEL
LIN {X 0,Y 263.203,Z 292.509,A -85,B 0,C 180,E1 -18380.318,E2 -18380.318} C_VEL
LIN {X 0,Y 263.124,Z 292.523,A -85,B 0,C 180,E1 -18385.307,E2 -18385.307} C_VEL
LIN {X 0,Y 263.106,Z 292.522,A -85,B 0,C 180,E1 -18386.672,E2 -18386.672} C_VEL
LIN {X 0,Y 262.481,Z 292.605,A -85,B 0,C 180,E1 -18387.949,E2 -18387.949} C_VEL
LIN {X 0,Y 259.639,Z 292.965,A -85,B 0,C 180,E1 -18390.03,E2 -18390.03} C_VEL
LIN {X 0,Y 257.199,Z 293.266,A -85,B 0,C 180,E1 -18391.723,E2 -18391.723} C_VEL
LIN {X 0,Y 256.15,Z 293.391,A -85,B 0,C 180,E1 -18393.037,E2 -18393.037} C_VEL
LIN {X 0,Y 256.066,Z 293.399,A -85,B 0,C 180,E1 -18393.482,E2 -18393.482} C_VEL
LIN {X 0,Y 256.12,Z 293.394,A -85,B 0,C 180,E1 -18397.278,E2 -18397.278} C_VEL
LIN {X 0,Y 256.022,Z 293.403,A -85,B 0,C 180,E1 -18401.217,E2 -18401.217} C_VEL
LIN {X 0,Y 256.024,Z 293.406,A -85,B 0,C 180,E1 -18405.546,E2 -18405.546} C_VEL
LIN {X 0,Y 256.024,Z 293.401,A -85,B 0,C 180,E1 -18408.795,E2 -18408.795} C_VEL
LIN {X 0,Y 256.109,Z 293.393,A -85,B 0,C 180,E1 -18412.868,E2 -18412.868} C_VEL
LIN {X 0,Y 256.076,Z 293.396,A -85,B 0,C 180,E1 -18416.712,E2 -18416.712} C_VEL
LIN {X 0,Y 256.065,Z 293.401,A -85,B 0,C 180,E1 -18420.398,E2 -18420.398} C_VEL
LIN {X 0,Y 256.353,Z 293.384,A -85,B 0,C 180,E1 -18423.877,E2 -18423.877} C_VEL
LIN {X 0,Y 257.457,Z 299.454,A -85,B 0,C 180,E1 -18426.26,E2 -18426.26} C_VEL
LIN {X 0,Y 256.64,Z 307.001,A -85,B 0,C 180,E1 -18429.148,E2 -18429.148} C_VEL
LIN {X 0,Y 255.877,Z 314.019,A -85,B 0,C 180,E1 -18431.797,E2 -18431.797} C_VEL
LIN {X 0,Y 256.616,Z 331.891,A -85,B 0,C 180,E1 -18432.629,E2 -18432.629} C_VEL
LIN {X 0,Y 258.297,Z 351.086,A -85,B 0,C 180,E1 -18433.517,E2 -18433.517} C_VEL
LIN {X 0,Y 257.278,Z 393.6,A -85,B 0,C 180,E1 -18435.518,E2 -18435.518} C_VEL
LIN {X 0,Y 256.858,Z 406.11,A -85,B 0,C 180,E1 -18436.454,E2 -18436.454} C_VEL
LIN {X 0,Y 256.304,Z 416.563,A -85,B 0,C 180,E1 -18437.532,E2 -18437.532} C_VEL
LIN {X 0,Y 255.779,Z 427.031,A -85,B 0,C 180,E1 -18438.914,E2 -18438.914} C_VEL
LIN {X 0,Y 255.41,Z 436.315,A -85,B 0,C 180,E1 -18440.5,E2 -18440.5} C_VEL
LIN {X 0,Y 255.052,Z 443.858,A -85,B 0,C 180,E1 -18442.084,E2 -18442.084} C_VEL
LIN {X 0,Y 254.928,Z 450.138,A -85,B 0,C 180,E1 -18443.672,E2 -18443.672} C_VEL
LIN {X 0,Y 254.739,Z 456.503,A -85,B 0,C 180,E1 -18445.652,E2 -18445.652} C_VEL
LIN {X 0,Y 254.588,Z 461.494,A -85,B 0,C 180,E1 -18447.63,E2 -18447.63} C_VEL
LIN {X 0,Y 254.659,Z 465.903,A -85,B 0,C 180,E1 -18450.003,E2 -18450.003} C_VEL
LIN {X 0,Y 254.228,Z 468.028,A -85,B 0,C 180,E1 -18451.587,E2 -18451.587} C_VEL
LIN {X 0,Y 254.16,Z 469.563,A -85,B 0,C 180,E1 -18453.173,E2 -18453.173} C_VEL
LIN {X 0,Y 254.155,Z 470.865,A -85,B 0,C 180,E1 -18455.396,E2 -18455.396} C_VEL
LIN {X 0,Y 254.586,Z 471.1,A -85,B 0,C 180,E1 -18457.936,E2 -18457.936} C_VEL
LIN {X 0,Y 255.096,Z 470.6,A -85,B 0,C 180,E1 -18459.517,E2 -18459.517} C_VEL
LIN {X 0,Y 255.87,Z 469.551,A -85,B 0,C 180,E1 -18461.088,E2 -18461.088} C_VEL
LIN {X 0,Y 257.472,Z 467.116,A -85,B 0,C 180,E1 -18463.418,E2 -18463.418} C_VEL
LIN {X 0,Y 259.68,Z 463.467,A -85,B 0,C 180,E1 -18465.705,E2 -18465.705} C_VEL
LIN {X 0,Y 262.143,Z 458.459,A -85,B 0,C 180,E1 -18467.96,E2 -18467.96} C_VEL
LIN {X 0,Y 264.703,Z 453.124,A -85,B 0,C 180,E1 -18469.789,E2 -18469.789} C_VEL
LIN {X 0,Y 267.722,Z 446.522,A -85,B 0,C 180,E1 -18471.565,E2 -18471.565} C_VEL
LIN {X 0,Y 270.361,Z 440.265,A -85,B 0,C 180,E1 -18472.952,E2 -18472.952} C_VEL
LIN {X 0,Y 273.983,Z 430.796,A -85,B 0,C 180,E1 -18474.637,E2 -18474.637} C_VEL
LIN {X 0,Y 277.21,Z 421.12,A -85,B 0,C 180,E1 -18475.936,E2 -18475.936} C_VEL
LIN {X 0,Y 280.272,Z 410.746,A -85,B 0,C 180,E1 -18477.035,E2 -18477.035} C_VEL
LIN {X 0,Y 283.376,Z 398.281,A -85,B 0,C 180,E1 -18478.015,E2 -18478.015} C_VEL
LIN {X 0,Y 285.386,Z 386.971,A -85,B 0,C 180,E1 -18478.685,E2 -18478.685} C_VEL
LIN {X 0,Y 288.601,Z 363.147,A -85,B 0,C 180,E1 -18479.808,E2 -18479.808} C_VEL
